RoboDK station: InvertedRobot.rdk

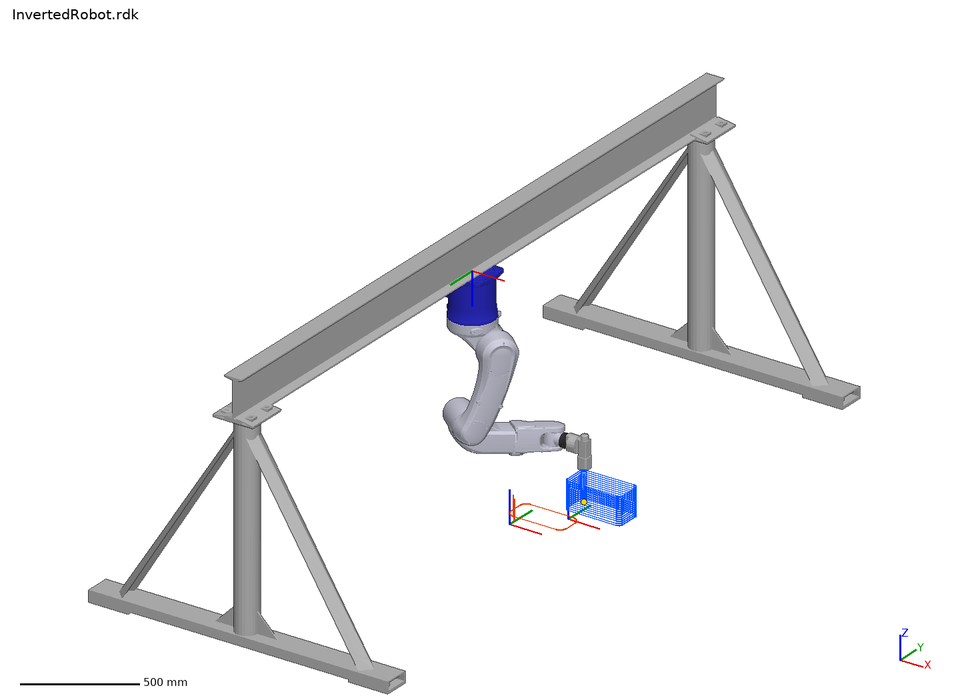
[picture v0: the station drawn from its stored meshes, robots at their saved joint values, targets as dots, program paths as lines]
Station InvertedRobot (saved by RoboDK 5.5.4). Poses are relative to the parent item; angles as X-Y-Z fixed-axis rotations.
Station parameters (name, value as stored): TAGS, ['Additive Manufacturing', 'Additive manufacturing']
  - frame Denso 1 at (0, -20, 974.25) mm, rotated rx -180 ry 0 rz 0 deg
    - robot Denso VS-6577G-B: 6 axes, payload 7 kg, reach 854 mm, repeatability 0.03 mm, weight 36 kg
        modified DH rows (alpha deg, a mm, theta deg, d mm): 0, 0, 0, 335; -90, 75, -90, 0; 0, 365, -90, 0; -90, 90, 0, 405; 90, 0, 0, 0; -90, 0, 0, 80
        joint limits [-170, -100, -119, -190, -120, -360] to [170, 135, 169, 190, 120, 360]; home [0, 0, 90, 0, 0, 0]; saved at [-52.91, -18.13, 101.16, 84.758, 53.229, -81.286]
      - tool nozzle, TCP at (110, 0, 80) mm, rotated rx 0 ry 90 rz 0 deg, size 158.8 x 76.2 x 114.9 mm, geometry from nozzle.STEP
  - frame Ref001 at (404.35, 97.88, -110) mm
    - object Part at (0, 0, 0) mm, size 120 x 120 x 160 mm, geometry from part.sld
  - machining project Print3D settings: C:/Users/silverBlacK/OneDrive - University of Idaho/Research/RoboticsResearch/WallSection.gcode | rotZ(0) | rotX(0)*rotY(0) | rotZ(0)
  - program Print3D1 (17608 instructions, listed below)
  - frame Ref002 at (374.35, -282.12, 10) mm
    - object Part at (0, 0, 0) mm, size 120 x 120 x 160 mm, geometry from part.sld
  - machining project Print3D settings: C:/Users/silverBlacK/OneDrive - University of Idaho/Research/RoboticsResearch/WallSections/12x12x0.875.gcode | rotZ(0) | rotX(0)*rotY(0) | rotz(0) | onStart | onPathStart | onApproach | onPoint | onRetract | onFinish | SetRPM(%1) | SetTool(%1) | Extruder(%1) | default | default | OutOnMov(%1) | OutOffMov(%1) | onPathFinish | M_RunCode(%1)
  - program Print3D (292 instructions, listed below)
  - Python program Extruder (listed below)
  - Python program SimulateFinalResult (listed below)
  - object GantryAssembly at (-570, -550, -380) mm, rotated rx 90 ry 0 rz 0 deg, size 1524 x 1270 x 3505.2 mm, geometry from GantryAssembly.STEP
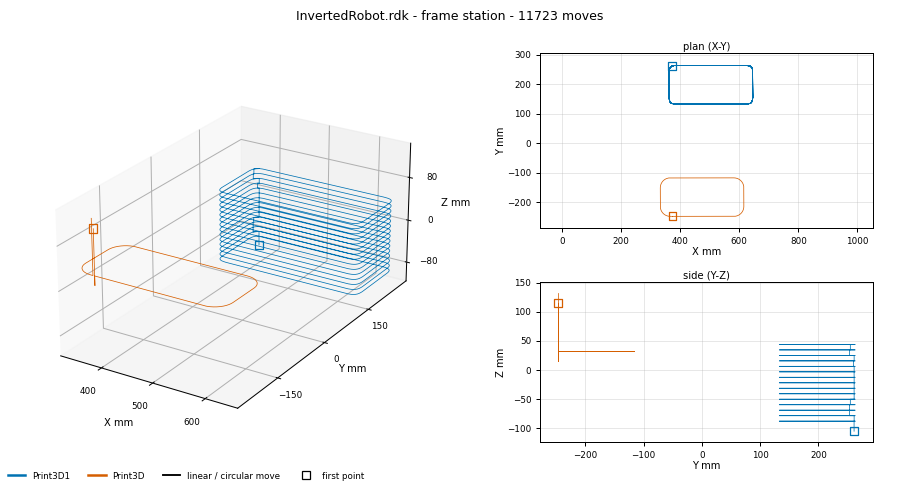
[picture p0: tool path of InvertedRobot.rdk in frame station, 11723 of 11723 moves have a stored position in this frame; points joined in program order, loops and branches not executed]

--- program Print3D1 (robot Denso VS-6577G-B) ---
  Smooth(1)
  Call M_RunCode(107)
  Call M_RunCode(104)
  Set speed (83.3 mm/s)
  Set speed (1000.0 mm/s)
  Set Ref.: Ref001
  Set Tool: nozzle
  Show nozzle
  MoveJ 1 to (-31.64, 163.21, 5) mm, rotated rx -180 ry 0 rz 180 deg; joints [-52.884, -5.749, 67.478, 70.281, 57.897, -56.003]
  MoveL 2 to (-31.64, 163.21, 5) mm, rotated rx -180 ry 0 rz 180 deg; joints [-52.884, -5.749, 67.478, 70.281, 57.897, -56.003]
  Call Extruder(-1)
  MoveL 3 to (-31.64, 163.21, 5) mm, rotated rx -180 ry 0 rz 180 deg; joints [-52.884, -5.749, 67.478, 70.281, 57.897, -56.003]
  Call M_RunCode(109)
  Call M_RunCode(82)
  Call Extruder(0.00000)
  Set speed (130.0 mm/s)
  MoveL 4 to (-31.64, 163.21, 22.23) mm, rotated rx 180 ry 0 rz -180 deg; joints [-52.884, -7.787, 72.321, 71.976, 56.989, -59.153]
  Call Extruder(-2.00000)
  Set speed (40.0 mm/s)
  MoveL 5 to (-31.64, 163.21, 22.23) mm, rotated rx 180 ry 0 rz -180 deg; joints [-52.884, -7.787, 72.321, 71.976, 56.989, -59.153]
  Call Extruder(0.00000)
  Set speed (130.0 mm/s)
  MoveL 6 to (-31.64, 163.21, 22.23) mm, rotated rx 180 ry 0 rz -180 deg; joints [-52.884, -7.787, 72.321, 71.976, 56.989, -59.153]
  Call Extruder(2.00000)
  Set speed (40.0 mm/s)
  MoveL 7 to (-31.64, 163.21, 22.23) mm, rotated rx 180 ry 0 rz -180 deg; joints [-52.884, -7.787, 72.321, 71.976, 56.989, -59.153]
  Set speed (30.0 mm/s)
  MoveL 8 to (-31.64, 163.21, 22.23) mm, rotated rx 180 ry 0 rz -180 deg; joints [-52.884, -7.787, 72.321, 71.976, 56.989, -59.153]
  Call Extruder(2.38024)
  MoveL 9 to (-31.93, 163.09, 22.22) mm, rotated rx 180 ry 0 rz 180 deg; joints [-52.91, -7.826, 72.354, 71.989, 57.013, -59.155]
  MoveL 10 to (-31.93, 163.09, 22.22) mm, rotated rx 180 ry 0 rz 180 deg; joints [-52.91, -7.826, 72.354, 71.989, 57.013, -59.155]
  Call Extruder(2.76227)
  MoveL 11 to (-32.22, 162.97, 22.22) mm, rotated rx 180 ry 0 rz -180 deg; joints [-52.936, -7.865, 72.387, 72.001, 57.037, -59.157]
  MoveL 12 to (-32.22, 162.97, 22.22) mm, rotated rx 180 ry 0 rz -180 deg; joints [-52.936, -7.865, 72.387, 72.001, 57.037, -59.157]
  Call Extruder(3.11872)
  MoveL 13 to (-32.49, 162.85, 22.22) mm, rotated rx -180 ry 0 rz 180 deg; joints [-52.96, -7.901, 72.418, 72.012, 57.06, -59.158]
  MoveL 14 to (-32.49, 162.85, 22.22) mm, rotated rx -180 ry 0 rz 180 deg; joints [-52.96, -7.901, 72.418, 72.012, 57.06, -59.158]
  Call Extruder(3.44932)
  MoveL 15 to (-32.74, 162.74, 22.22) mm, rotated rx 180 ry 0 rz 180 deg; joints [-52.982, -7.935, 72.446, 72.022, 57.08, -59.16]
  MoveL 16 to (-32.74, 162.74, 22.22) mm, rotated rx 180 ry 0 rz 180 deg; joints [-52.982, -7.935, 72.446, 72.022, 57.08, -59.16]
  Call Extruder(3.78134)
  MoveL 17 to (-32.99, 162.64, 22.22) mm, rotated rx -180 ry 0 rz 180 deg; joints [-53.004, -7.968, 72.475, 72.032, 57.1, -59.161]
  MoveL 18 to (-32.99, 162.64, 22.22) mm, rotated rx -180 ry 0 rz 180 deg; joints [-53.004, -7.968, 72.475, 72.032, 57.1, -59.161]
  Call Extruder(4.21321)
  MoveL 19 to (-33.29, 162.46, 22.22) mm, rotated rx -180 ry 0 rz 180 deg; joints [-53.026, -8.015, 72.514, 72.042, 57.122, -59.16]
  MoveL 20 to (-33.29, 162.46, 22.22) mm, rotated rx -180 ry 0 rz 180 deg; joints [-53.026, -8.015, 72.514, 72.042, 57.122, -59.16]
  Call Extruder(4.64692)
  MoveL 21 to (-33.6, 162.29, 22.22) mm, rotated rx 180 ry 0 rz 180 deg; joints [-53.049, -8.061, 72.553, 72.051, 57.143, -59.16]
  MoveL 22 to (-33.6, 162.29, 22.22) mm, rotated rx 180 ry 0 rz 180 deg; joints [-53.049, -8.061, 72.553, 72.051, 57.143, -59.16]
  Call Extruder(5.08247)
  MoveL 23 to (-33.9, 162.11, 22.23) mm, rotated rx 180 ry 0 rz 180 deg; joints [-53.071, -8.107, 72.591, 72.06, 57.165, -59.159]
  MoveL 24 to (-33.9, 162.11, 22.23) mm, rotated rx 180 ry 0 rz 180 deg; joints [-53.071, -8.107, 72.591, 72.06, 57.165, -59.159]
  Call Extruder(5.51986)
  MoveL 25 to (-34.21, 161.94, 22.22) mm, rotated rx 180 ry 0 rz 180 deg; joints [-53.094, -8.153, 72.63, 72.07, 57.186, -59.158]
  MoveL 26 to (-34.21, 161.94, 22.22) mm, rotated rx 180 ry 0 rz 180 deg; joints [-53.094, -8.153, 72.63, 72.07, 57.186, -59.158]
  Call Extruder(5.89660)
  MoveL 27 to (-34.45, 161.76, 22.22) mm, rotated rx 180 ry 0 rz 180 deg; joints [-53.109, -8.194, 72.665, 72.075, 57.201, -59.156]
  MoveL 28 to (-34.45, 161.76, 22.22) mm, rotated rx 180 ry 0 rz 180 deg; joints [-53.109, -8.194, 72.665, 72.075, 57.201, -59.156]
  Call Extruder(6.59657)
  MoveL 29 to (-34.9, 161.43, 22.23) mm, rotated rx 180 ry 0 rz 180 deg; joints [-53.135, -8.27, 72.728, 72.084, 57.228, -59.151]
  MoveL 30 to (-34.9, 161.43, 22.23) mm, rotated rx 180 ry 0 rz 180 deg; joints [-53.135, -8.27, 72.728, 72.084, 57.228, -59.151]
  Call Extruder(7.29934)
  MoveL 31 to (-35.35, 161.1, 22.22) mm, rotated rx 180 ry 0 rz 180 deg; joints [-53.163, -8.346, 72.792, 72.093, 57.255, -59.146]
  Call Extruder(9.03811)
  MoveL 32 to (-36.39, 160.19, 22.22) mm, rotated rx 180 ry 0 rz 180 deg; joints [-53.209, -8.538, 72.953, 72.102, 57.305, -59.126]
  Call Extruder(10.77694)
  MoveL 33 to (-37.3, 159.15, 22.22) mm, rotated rx 180 ry 0 rz 180 deg; joints [-53.227, -8.733, 73.115, 72.093, 57.33, -59.094]
  Call Extruder(11.12832)
  MoveL 34 to (-37.47, 158.93, 22.22) mm, rotated rx 180 ry 0 rz -180 deg; joints [-53.227, -8.773, 73.148, 72.088, 57.332, -59.087]
  MoveL 35 to (-37.47, 158.93, 22.22) mm, rotated rx 180 ry 0 rz -180 deg; joints [-53.227, -8.773, 73.148, 72.088, 57.332, -59.087]
  Call Extruder(11.82828)
  MoveL 36 to (-37.79, 158.48, 22.22) mm, rotated rx 180 ry 0 rz 180 deg; joints [-53.226, -8.852, 73.214, 72.079, 57.335, -59.071]
  MoveL 37 to (-37.79, 158.48, 22.22) mm, rotated rx 180 ry 0 rz 180 deg; joints [-53.226, -8.852, 73.214, 72.079, 57.335, -59.071]
  Call Extruder(12.52544)
  MoveL 38 to (-38.12, 158.03, 22.22) mm, rotated rx 180 ry 0 rz 180 deg; joints [-53.224, -8.931, 73.279, 72.07, 57.338, -59.055]
  MoveL 39 to (-38.12, 158.03, 22.22) mm, rotated rx 180 ry 0 rz 180 deg; joints [-53.224, -8.931, 73.279, 72.07, 57.338, -59.055]
  Call Extruder(12.77229)
  MoveL 40 to (-38.22, 157.85, 22.22) mm, rotated rx -180 ry 0 rz 180 deg; joints [-53.221, -8.959, 73.302, 72.065, 57.336, -59.048]
  MoveL 41 to (-38.22, 157.85, 22.22) mm, rotated rx -180 ry 0 rz 180 deg; joints [-53.221, -8.959, 73.302, 72.065, 57.336, -59.048]
  Call Extruder(13.20785)
  MoveL 42 to (-38.4, 157.55, 22.22) mm, rotated rx 180 ry 0 rz 180 deg; joints [-53.214, -9.008, 73.343, 72.055, 57.333, -59.036]
  MoveL 43 to (-38.4, 157.55, 22.22) mm, rotated rx 180 ry 0 rz 180 deg; joints [-53.214, -9.008, 73.343, 72.055, 57.333, -59.036]
  Call Extruder(13.64157)
  MoveL 44 to (-38.57, 157.25, 22.22) mm, rotated rx -180 ry 0 rz 180 deg; joints [-53.207, -9.057, 73.383, 72.046, 57.33, -59.024]
  MoveL 45 to (-38.57, 157.25, 22.22) mm, rotated rx -180 ry 0 rz 180 deg; joints [-53.207, -9.057, 73.383, 72.046, 57.33, -59.024]
  Call Extruder(14.07344)
  MoveL 46 to (-38.75, 156.94, 22.22) mm, rotated rx 180 ry 0 rz 180 deg; joints [-53.2, -9.106, 73.424, 72.036, 57.327, -59.012]
  MoveL 47 to (-38.75, 156.94, 22.22) mm, rotated rx 180 ry 0 rz 180 deg; joints [-53.2, -9.106, 73.424, 72.036, 57.327, -59.012]
  Call Extruder(14.45383)
  MoveL 48 to (-38.89, 156.67, 22.22) mm, rotated rx 180 ry 0 rz 180 deg; joints [-53.191, -9.15, 73.459, 72.026, 57.322, -59.001]
  MoveL 49 to (-38.89, 156.67, 22.22) mm, rotated rx 180 ry 0 rz 180 deg; joints [-53.191, -9.15, 73.459, 72.026, 57.322, -59.001]
  Call Extruder(14.78446)
  MoveL 50 to (-39, 156.42, 22.22) mm, rotated rx 180 ry 0 rz 180 deg; joints [-53.18, -9.187, 73.49, 72.016, 57.314, -58.99]
  MoveL 51 to (-39, 156.42, 22.22) mm, rotated rx 180 ry 0 rz 180 deg; joints [-53.18, -9.187, 73.49, 72.016, 57.314, -58.99]
  Call Extruder(15.11366)
  MoveL 52 to (-39.11, 156.17, 22.22) mm, rotated rx 180 ry 0 rz 180 deg; joints [-53.17, -9.224, 73.52, 72.005, 57.307, -58.979]
  MoveL 53 to (-39.11, 156.17, 22.22) mm, rotated rx 180 ry 0 rz 180 deg; joints [-53.17, -9.224, 73.52, 72.005, 57.307, -58.979]
  Call Extruder(15.49565)
  MoveL 54 to (-39.23, 155.88, 22.22) mm, rotated rx 180 ry 0 rz 180 deg; joints [-53.156, -9.267, 73.556, 71.992, 57.298, -58.965]
  MoveL 55 to (-39.23, 155.88, 22.22) mm, rotated rx 180 ry 0 rz 180 deg; joints [-53.156, -9.267, 73.556, 71.992, 57.298, -58.965]
  Call Extruder(15.87585)
  MoveL 56 to (-39.35, 155.58, 22.22) mm, rotated rx 180 ry 0 rz 180 deg; joints [-53.143, -9.31, 73.591, 71.98, 57.29, -58.952]
  MoveL 57 to (-39.35, 155.58, 22.22) mm, rotated rx 180 ry 0 rz 180 deg; joints [-53.143, -9.31, 73.591, 71.98, 57.29, -58.952]
  Call Extruder(16.18353)
  MoveL 58 to (-39.44, 155.34, 22.23) mm, rotated rx 180 ry 0 rz 180 deg; joints [-53.131, -9.345, 73.619, 71.968, 57.281, -58.941]
  MoveL 59 to (-39.44, 155.34, 22.23) mm, rotated rx 180 ry 0 rz 180 deg; joints [-53.131, -9.345, 73.619, 71.968, 57.281, -58.941]
  Call Extruder(16.41988)
  MoveL 60 to (-39.5, 155.15, 22.22) mm, rotated rx 180 ry 0 rz 180 deg; joints [-53.121, -9.371, 73.641, 71.959, 57.274, -58.932]
  MoveL 61 to (-39.5, 155.15, 22.22) mm, rotated rx 180 ry 0 rz 180 deg; joints [-53.121, -9.371, 73.641, 71.959, 57.274, -58.932]
  Call Extruder(16.65518)
  MoveL 62 to (-39.56, 154.97, 22.23) mm, rotated rx 180 ry 0 rz 180 deg; joints [-53.11, -9.398, 73.663, 71.949, 57.266, -58.923]
  MoveL 63 to (-39.56, 154.97, 22.23) mm, rotated rx 180 ry 0 rz 180 deg; joints [-53.11, -9.398, 73.663, 71.949, 57.266, -58.923]
  Call Extruder(16.88943)
  MoveL 64 to (-39.62, 154.78, 22.22) mm, rotated rx 180 ry 0 rz 180 deg; joints [-53.099, -9.424, 73.684, 71.94, 57.258, -58.914]
  MoveL 65 to (-39.62, 154.78, 22.22) mm, rotated rx 180 ry 0 rz 180 deg; joints [-53.099, -9.424, 73.684, 71.94, 57.258, -58.914]
  Call Extruder(17.12262)
  MoveL 66 to (-39.68, 154.59, 22.22) mm, rotated rx 180 ry 0 rz -180 deg; joints [-53.088, -9.45, 73.706, 71.93, 57.25, -58.905]
  MoveL 67 to (-39.68, 154.59, 22.22) mm, rotated rx 180 ry 0 rz -180 deg; joints [-53.088, -9.45, 73.706, 71.93, 57.25, -58.905]
  Call Extruder(17.37548)
  MoveL 68 to (-39.75, 154.38, 22.23) mm, rotated rx 180 ry 0 rz 180 deg; joints [-53.076, -9.479, 73.729, 71.919, 57.242, -58.895]
  MoveL 69 to (-39.75, 154.38, 22.23) mm, rotated rx 180 ry 0 rz 180 deg; joints [-53.076, -9.479, 73.729, 71.919, 57.242, -58.895]
  Call Extruder(17.64775)
  MoveL 70 to (-39.81, 154.16, 22.23) mm, rotated rx 180 ry 0 rz 180 deg; joints [-53.063, -9.51, 73.754, 71.908, 57.232, -58.884]
  MoveL 71 to (-39.81, 154.16, 22.23) mm, rotated rx 180 ry 0 rz 180 deg; joints [-53.063, -9.51, 73.754, 71.908, 57.232, -58.884]
  Call Extruder(17.91868)
  MoveL 72 to (-39.88, 153.94, 22.22) mm, rotated rx 180 ry 0 rz 180 deg; joints [-53.049, -9.541, 73.779, 71.896, 57.222, -58.873]
  MoveL 73 to (-39.88, 153.94, 22.22) mm, rotated rx 180 ry 0 rz 180 deg; joints [-53.049, -9.541, 73.779, 71.896, 57.222, -58.873]
  Call Extruder(18.18828)
  MoveL 74 to (-39.95, 153.71, 22.23) mm, rotated rx 180 ry 0 rz 180 deg; joints [-53.036, -9.572, 73.804, 71.884, 57.212, -58.862]
  MoveL 75 to (-39.95, 153.71, 22.23) mm, rotated rx 180 ry 0 rz 180 deg; joints [-53.036, -9.572, 73.804, 71.884, 57.212, -58.862]
  Call Extruder(18.45654)
  MoveL 76 to (-40.02, 153.49, 22.23) mm, rotated rx 180 ry 0 rz 180 deg; joints [-53.022, -9.602, 73.829, 71.872, 57.202, -58.851]
  MoveL 77 to (-40.02, 153.49, 22.23) mm, rotated rx 180 ry 0 rz 180 deg; joints [-53.022, -9.602, 73.829, 71.872, 57.202, -58.851]
  Call Extruder(18.69554)
  MoveL 78 to (-40.06, 153.28, 22.23) mm, rotated rx 180 ry 0 rz 180 deg; joints [-53.007, -9.629, 73.851, 71.86, 57.191, -58.841]
  MoveL 79 to (-40.06, 153.28, 22.23) mm, rotated rx 180 ry 0 rz 180 deg; joints [-53.007, -9.629, 73.851, 71.86, 57.191, -58.841]
  Call Extruder(18.93348)
  MoveL 80 to (-40.11, 153.08, 22.22) mm, rotated rx -180 ry 0 rz 180 deg; joints [-52.993, -9.656, 73.873, 71.848, 57.18, -58.83]
  MoveL 81 to (-40.11, 153.08, 22.22) mm, rotated rx -180 ry 0 rz 180 deg; joints [-52.993, -9.656, 73.873, 71.848, 57.18, -58.83]
  Call Extruder(19.17035)
  MoveL 82 to (-40.15, 152.88, 22.23) mm, rotated rx 180 ry 0 rz 180 deg; joints [-52.978, -9.682, 73.894, 71.836, 57.169, -58.819]
  MoveL 83 to (-40.15, 152.88, 22.23) mm, rotated rx 180 ry 0 rz 180 deg; joints [-52.978, -9.682, 73.894, 71.836, 57.169, -58.819]
  Call Extruder(19.40615)
  MoveL 84 to (-40.2, 152.67, 22.23) mm, rotated rx 180 ry 0 rz 180 deg; joints [-52.963, -9.709, 73.916, 71.824, 57.158, -58.809]
  MoveL 85 to (-40.2, 152.67, 22.23) mm, rotated rx 180 ry 0 rz 180 deg; joints [-52.963, -9.709, 73.916, 71.824, 57.158, -58.809]
  Call Extruder(19.66605)
  MoveL 86 to (-40.24, 152.45, 22.23) mm, rotated rx 180 ry 0 rz 180 deg; joints [-52.946, -9.738, 73.94, 71.81, 57.146, -58.797]
  MoveL 87 to (-40.24, 152.45, 22.23) mm, rotated rx 180 ry 0 rz 180 deg; joints [-52.946, -9.738, 73.94, 71.81, 57.146, -58.797]
  Call Extruder(19.94972)
  MoveL 88 to (-40.29, 152.2, 22.22) mm, rotated rx 180 ry 0 rz 180 deg; joints [-52.928, -9.77, 73.966, 71.795, 57.132, -58.784]
  MoveL 89 to (-40.29, 152.2, 22.22) mm, rotated rx 180 ry 0 rz 180 deg; joints [-52.928, -9.77, 73.966, 71.795, 57.132, -58.784]
  Call Extruder(20.23193)
  MoveL 90 to (-40.34, 151.95, 22.22) mm, rotated rx 180 ry 0 rz 180 deg; joints [-52.909, -9.803, 73.992, 71.779, 57.117, -58.77]
  MoveL 91 to (-40.34, 151.95, 22.22) mm, rotated rx 180 ry 0 rz 180 deg; joints [-52.909, -9.803, 73.992, 71.779, 57.117, -58.77]
  Call Extruder(20.51271)
  MoveL 92 to (-40.39, 151.7, 22.23) mm, rotated rx 180 ry 0 rz 180 deg; joints [-52.89, -9.835, 74.018, 71.764, 57.103, -58.757]
  MoveL 93 to (-40.39, 151.7, 22.23) mm, rotated rx 180 ry 0 rz 180 deg; joints [-52.89, -9.835, 74.018, 71.764, 57.103, -58.757]
  Call Extruder(20.79205)
  MoveL 94 to (-40.44, 151.45, 22.22) mm, rotated rx 180 ry 0 rz -180 deg; joints [-52.871, -9.867, 74.043, 71.748, 57.089, -58.744]
  MoveL 95 to (-40.44, 151.45, 22.22) mm, rotated rx 180 ry 0 rz -180 deg; joints [-52.871, -9.867, 74.043, 71.748, 57.089, -58.744]
  Call Extruder(21.06994)
  MoveL 96 to (-40.49, 151.2, 22.22) mm, rotated rx 180 ry 0 rz 180 deg; joints [-52.853, -9.899, 74.069, 71.733, 57.075, -58.731]
  MoveL 97 to (-40.49, 151.2, 22.22) mm, rotated rx 180 ry 0 rz 180 deg; joints [-52.853, -9.899, 74.069, 71.733, 57.075, -58.731]
  Call Extruder(21.34639)
  MoveL 98 to (-40.54, 150.95, 22.23) mm, rotated rx 180 ry 0 rz 180 deg; joints [-52.834, -9.93, 74.095, 71.718, 57.061, -58.717]
  MoveL 99 to (-40.54, 150.95, 22.23) mm, rotated rx 180 ry 0 rz 180 deg; joints [-52.834, -9.93, 74.095, 71.718, 57.061, -58.717]
  Call Extruder(21.65140)
  MoveL 100 to (-40.59, 150.67, 22.22) mm, rotated rx 180 ry 0 rz 180 deg; joints [-52.812, -9.966, 74.123, 71.7, 57.044, -58.702]
  MoveL 101 to (-40.59, 150.67, 22.22) mm, rotated rx 180 ry 0 rz 180 deg; joints [-52.812, -9.966, 74.123, 71.7, 57.044, -58.702]
  Call Extruder(21.98479)
  MoveL 102 to (-40.64, 150.37, 22.22) mm, rotated rx -180 ry 0 rz 180 deg; joints [-52.787, -10.004, 74.154, 71.68, 57.025, -58.686]
  MoveL 103 to (-40.64, 150.37, 22.22) mm, rotated rx -180 ry 0 rz 180 deg; joints [-52.787, -10.004, 74.154, 71.68, 57.025, -58.686]
  Call Extruder(22.31647)
  MoveL 104 to (-40.69, 150.06, 22.22) mm, rotated rx 180 ry 0 rz 180 deg; joints [-52.762, -10.042, 74.185, 71.66, 57.006, -58.669]
  MoveL 105 to (-40.69, 150.06, 22.22) mm, rotated rx 180 ry 0 rz 180 deg; joints [-52.762, -10.042, 74.185, 71.66, 57.006, -58.669]
  Call Extruder(22.64643)
  MoveL 106 to (-40.74, 149.76, 22.22) mm, rotated rx -180 ry 0 rz 180 deg; joints [-52.737, -10.08, 74.215, 71.64, 56.988, -58.652]
  MoveL 107 to (-40.74, 149.76, 22.22) mm, rotated rx -180 ry 0 rz 180 deg; joints [-52.737, -10.08, 74.215, 71.64, 56.988, -58.652]
  Call Extruder(22.97467)
  MoveL 108 to (-40.78, 149.45, 22.23) mm, rotated rx 180 ry 0 rz 180 deg; joints [-52.712, -10.118, 74.246, 71.62, 56.969, -58.635]
  MoveL 109 to (-40.78, 149.45, 22.23) mm, rotated rx 180 ry 0 rz 180 deg; joints [-52.712, -10.118, 74.246, 71.62, 56.969, -58.635]
  Call Extruder(23.30119)
  MoveL 110 to (-40.83, 149.14, 22.22) mm, rotated rx 180 ry 0 rz -180 deg; joints [-52.687, -10.156, 74.277, 71.6, 56.95, -58.618]
  MoveL 111 to (-40.83, 149.14, 22.22) mm, rotated rx 180 ry 0 rz -180 deg; joints [-52.687, -10.156, 74.277, 71.6, 56.95, -58.618]
  Call Extruder(23.66827)
  MoveL 112 to (-40.88, 148.8, 22.23) mm, rotated rx 180 ry 0 rz -180 deg; joints [-52.658, -10.199, 74.311, 71.576, 56.927, -58.598]
  MoveL 113 to (-40.88, 148.8, 22.23) mm, rotated rx 180 ry 0 rz -180 deg; joints [-52.658, -10.199, 74.311, 71.576, 56.927, -58.598]
  Call Extruder(24.07571)
  MoveL 114 to (-40.92, 148.41, 22.22) mm, rotated rx 180 ry 0 rz 180 deg; joints [-52.624, -10.246, 74.348, 71.549, 56.901, -58.576]
  MoveL 115 to (-40.92, 148.41, 22.22) mm, rotated rx 180 ry 0 rz 180 deg; joints [-52.624, -10.246, 74.348, 71.549, 56.901, -58.576]
  Call Extruder(24.48110)
  MoveL 116 to (-40.97, 148.02, 22.22) mm, rotated rx 180 ry 0 rz 180 deg; joints [-52.59, -10.292, 74.386, 71.522, 56.875, -58.554]
  MoveL 117 to (-40.97, 148.02, 22.22) mm, rotated rx 180 ry 0 rz 180 deg; joints [-52.59, -10.292, 74.386, 71.522, 56.875, -58.554]
  Call Extruder(24.88445)
  MoveL 118 to (-41.02, 147.63, 22.22) mm, rotated rx -180 ry 0 rz 180 deg; joints [-52.556, -10.339, 74.423, 71.495, 56.849, -58.532]
  MoveL 119 to (-41.02, 147.63, 22.22) mm, rotated rx -180 ry 0 rz 180 deg; joints [-52.556, -10.339, 74.423, 71.495, 56.849, -58.532]
  Call Extruder(25.28574)
  MoveL 120 to (-41.06, 147.25, 22.22) mm, rotated rx 180 ry 0 rz 180 deg; joints [-52.521, -10.386, 74.46, 71.468, 56.823, -58.51]
  MoveL 121 to (-41.06, 147.25, 22.22) mm, rotated rx 180 ry 0 rz 180 deg; joints [-52.521, -10.386, 74.46, 71.468, 56.823, -58.51]
  Call Extruder(25.89062)
  MoveL 122 to (-41.11, 146.66, 22.23) mm, rotated rx 180 ry 0 rz 180 deg; joints [-52.466, -10.455, 74.515, 71.425, 56.78, -58.475]
  MoveL 123 to (-41.11, 146.66, 22.23) mm, rotated rx 180 ry 0 rz 180 deg; joints [-52.466, -10.455, 74.515, 71.425, 56.78, -58.475]
  Call Extruder(26.49235)
  MoveL 124 to (-41.15, 146.07, 22.22) mm, rotated rx 180 ry 0 rz 180 deg; joints [-52.411, -10.524, 74.57, 71.381, 56.737, -58.44]
  MoveL 125 to (-41.15, 146.07, 22.22) mm, rotated rx 180 ry 0 rz 180 deg; joints [-52.411, -10.524, 74.57, 71.381, 56.737, -58.44]
  Call Extruder(27.09093)
  MoveL 126 to (-41.2, 145.48, 22.22) mm, rotated rx -180 ry 0 rz 180 deg; joints [-52.355, -10.593, 74.625, 71.338, 56.695, -58.404]
  MoveL 127 to (-41.2, 145.48, 22.22) mm, rotated rx -180 ry 0 rz 180 deg; joints [-52.355, -10.593, 74.625, 71.338, 56.695, -58.404]
  Call Extruder(28.26271)
  MoveL 128 to (-41.25, 144.32, 22.22) mm, rotated rx 180 ry 0 rz 180 deg; joints [-52.239, -10.724, 74.729, 71.247, 56.604, -58.333]
  MoveL 129 to (-41.25, 144.32, 22.22) mm, rotated rx 180 ry 0 rz 180 deg; joints [-52.239, -10.724, 74.729, 71.247, 56.604, -58.333]
  Call Extruder(29.72057)
  MoveL 130 to (-41.29, 142.86, 22.22) mm, rotated rx -180 ry 0 rz 180 deg; joints [-52.09, -10.887, 74.858, 71.132, 56.489, -58.243]
  Call Extruder(115.61408)
  MoveL 131 to (-41.29, 57.14, 22.22) mm, rotated rx 180 ry 0 rz 180 deg; joints [-40.759, -19.184, 80.692, 61.037, 48.262, -50.261]
  Call Extruder(116.48916)
  MoveL 132 to (-41.27, 56.26, 22.22) mm, rotated rx 180 ry 0 rz -180 deg; joints [-40.614, -19.255, 80.736, 60.892, 48.164, -50.147]
  MoveL 133 to (-41.27, 56.26, 22.22) mm, rotated rx 180 ry 0 rz -180 deg; joints [-40.614, -19.255, 80.736, 60.892, 48.164, -50.147]
  Call Extruder(117.66094)
  MoveL 134 to (-41.23, 55.1, 22.22) mm, rotated rx -180 ry 0 rz 180 deg; joints [-40.419, -19.347, 80.792, 60.696, 48.032, -49.993]
  MoveL 135 to (-41.23, 55.1, 22.22) mm, rotated rx -180 ry 0 rz 180 deg; joints [-40.419, -19.347, 80.792, 60.696, 48.032, -49.993]
  Call Extruder(118.54904)
  MoveL 136 to (-41.18, 54.23, 22.22) mm, rotated rx -180 ry 0 rz 180 deg; joints [-40.269, -19.414, 80.834, 60.545, 47.93, -49.875]
  MoveL 137 to (-41.18, 54.23, 22.22) mm, rotated rx -180 ry 0 rz 180 deg; joints [-40.269, -19.414, 80.834, 60.545, 47.93, -49.875]
  Call Extruder(119.15077)
  MoveL 138 to (-41.13, 53.64, 22.23) mm, rotated rx -180 ry 0 rz 180 deg; joints [-40.165, -19.458, 80.86, 60.442, 47.859, -49.794]
  MoveL 139 to (-41.13, 53.64, 22.23) mm, rotated rx -180 ry 0 rz 180 deg; joints [-40.165, -19.458, 80.86, 60.442, 47.859, -49.794]
  Call Extruder(119.75565)
  MoveL 140 to (-41.09, 53.05, 22.22) mm, rotated rx 180 ry 0 rz 180 deg; joints [-40.062, -19.502, 80.887, 60.338, 47.788, -49.714]
  MoveL 141 to (-41.09, 53.05, 22.22) mm, rotated rx 180 ry 0 rz 180 deg; joints [-40.062, -19.502, 80.887, 60.338, 47.788, -49.714]
  Call Extruder(120.26021)
  MoveL 142 to (-41.04, 52.56, 22.22) mm, rotated rx 180 ry 0 rz 180 deg; joints [-39.975, -19.538, 80.909, 60.251, 47.729, -49.646]
  MoveL 143 to (-41.04, 52.56, 22.22) mm, rotated rx 180 ry 0 rz 180 deg; joints [-39.975, -19.538, 80.909, 60.251, 47.729, -49.646]
  Call Extruder(120.66355)
  MoveL 144 to (-40.99, 52.17, 22.22) mm, rotated rx 180 ry 0 rz -180 deg; joints [-39.904, -19.565, 80.925, 60.181, 47.68, -49.592]
  MoveL 145 to (-40.99, 52.17, 22.22) mm, rotated rx 180 ry 0 rz -180 deg; joints [-39.904, -19.565, 80.925, 60.181, 47.68, -49.592]
  Call Extruder(121.06894)
  MoveL 146 to (-40.95, 51.78, 22.23) mm, rotated rx -180 ry 0 rz 180 deg; joints [-39.833, -19.592, 80.942, 60.111, 47.632, -49.538]
  MoveL 147 to (-40.95, 51.78, 22.23) mm, rotated rx -180 ry 0 rz 180 deg; joints [-39.833, -19.592, 80.942, 60.111, 47.632, -49.538]
  Call Extruder(121.47639)
  MoveL 148 to (-40.9, 51.4, 22.22) mm, rotated rx 180 ry 0 rz 180 deg; joints [-39.763, -19.619, 80.958, 60.04, 47.583, -49.484]
  MoveL 149 to (-40.9, 51.4, 22.22) mm, rotated rx 180 ry 0 rz 180 deg; joints [-39.763, -19.619, 80.958, 60.04, 47.583, -49.484]
  Call Extruder(121.88588)
  MoveL 150 to (-40.86, 51.01, 22.22) mm, rotated rx -180 ry 0 rz 180 deg; joints [-39.692, -19.646, 80.975, 59.969, 47.535, -49.429]
  MoveL 151 to (-40.86, 51.01, 22.22) mm, rotated rx -180 ry 0 rz 180 deg; joints [-39.692, -19.646, 80.975, 59.969, 47.535, -49.429]
  Call Extruder(122.21240)
  MoveL 152 to (-40.81, 50.7, 22.22) mm, rotated rx -180 ry 0 rz 180 deg; joints [-39.634, -19.666, 80.987, 59.912, 47.495, -49.386]
  MoveL 153 to (-40.81, 50.7, 22.22) mm, rotated rx -180 ry 0 rz 180 deg; joints [-39.634, -19.666, 80.987, 59.912, 47.495, -49.386]
  Call Extruder(122.54064)
  MoveL 154 to (-40.76, 50.4, 22.22) mm, rotated rx 180 ry 0 rz -180 deg; joints [-39.576, -19.686, 80.999, 59.854, 47.455, -49.342]
  MoveL 155 to (-40.76, 50.4, 22.22) mm, rotated rx 180 ry 0 rz -180 deg; joints [-39.576, -19.686, 80.999, 59.854, 47.455, -49.342]
  Call Extruder(122.87060)
  MoveL 156 to (-40.71, 50.09, 22.23) mm, rotated rx 180 ry 0 rz 180 deg; joints [-39.518, -19.706, 81.011, 59.797, 47.415, -49.298]
  MoveL 157 to (-40.71, 50.09, 22.23) mm, rotated rx 180 ry 0 rz 180 deg; joints [-39.518, -19.706, 81.011, 59.797, 47.415, -49.298]
  Call Extruder(123.20228)
  MoveL 158 to (-40.66, 49.79, 22.23) mm, rotated rx -180 ry 0 rz 180 deg; joints [-39.46, -19.726, 81.023, 59.74, 47.375, -49.254]
  MoveL 159 to (-40.66, 49.79, 22.23) mm, rotated rx -180 ry 0 rz 180 deg; joints [-39.46, -19.726, 81.023, 59.74, 47.375, -49.254]
  Call Extruder(123.53568)
  MoveL 160 to (-40.61, 49.48, 22.22) mm, rotated rx 180 ry 0 rz 180 deg; joints [-39.402, -19.746, 81.035, 59.682, 47.335, -49.21]
  MoveL 161 to (-40.61, 49.48, 22.22) mm, rotated rx 180 ry 0 rz 180 deg; joints [-39.402, -19.746, 81.035, 59.682, 47.335, -49.21]
  Call Extruder(123.87079)
  MoveL 162 to (-40.57, 49.17, 22.22) mm, rotated rx -180 ry 0 rz 180 deg; joints [-39.344, -19.765, 81.047, 59.624, 47.295, -49.166]
  MoveL 163 to (-40.57, 49.17, 22.22) mm, rotated rx -180 ry 0 rz 180 deg; joints [-39.344, -19.765, 81.047, 59.624, 47.295, -49.166]
  Call Extruder(124.14680)
  MoveL 164 to (-40.52, 48.93, 22.23) mm, rotated rx 180 ry 0 rz 180 deg; joints [-39.296, -19.781, 81.056, 59.576, 47.262, -49.129]
  MoveL 165 to (-40.52, 48.93, 22.23) mm, rotated rx 180 ry 0 rz 180 deg; joints [-39.296, -19.781, 81.056, 59.576, 47.262, -49.129]
  Call Extruder(124.42424)
  MoveL 166 to (-40.47, 48.68, 22.22) mm, rotated rx 180 ry 0 rz 180 deg; joints [-39.247, -19.796, 81.065, 59.528, 47.228, -49.093]
  MoveL 167 to (-40.47, 48.68, 22.22) mm, rotated rx 180 ry 0 rz 180 deg; joints [-39.247, -19.796, 81.065, 59.528, 47.228, -49.093]
  Call Extruder(124.70312)
  MoveL 168 to (-40.42, 48.43, 22.23) mm, rotated rx 180 ry 0 rz 180 deg; joints [-39.198, -19.811, 81.074, 59.479, 47.194, -49.056]
  MoveL 169 to (-40.42, 48.43, 22.23) mm, rotated rx 180 ry 0 rz 180 deg; joints [-39.198, -19.811, 81.074, 59.479, 47.194, -49.056]
  Call Extruder(124.98344)
  MoveL 170 to (-40.37, 48.18, 22.23) mm, rotated rx -180 ry 0 rz 180 deg; joints [-39.149, -19.826, 81.083, 59.431, 47.16, -49.019]
  MoveL 171 to (-40.37, 48.18, 22.23) mm, rotated rx -180 ry 0 rz 180 deg; joints [-39.149, -19.826, 81.083, 59.431, 47.16, -49.019]
  Call Extruder(125.26519)
  MoveL 172 to (-40.32, 47.93, 22.22) mm, rotated rx -180 ry 0 rz -180 deg; joints [-39.101, -19.841, 81.093, 59.382, 47.126, -48.983]
  MoveL 173 to (-40.32, 47.93, 22.22) mm, rotated rx -180 ry 0 rz -180 deg; joints [-39.101, -19.841, 81.093, 59.382, 47.126, -48.983]
  Call Extruder(125.54838)
  MoveL 174 to (-40.27, 47.68, 22.22) mm, rotated rx 180 ry 0 rz 180 deg; joints [-39.052, -19.856, 81.102, 59.334, 47.092, -48.946]
  MoveL 175 to (-40.27, 47.68, 22.22) mm, rotated rx 180 ry 0 rz 180 deg; joints [-39.052, -19.856, 81.102, 59.334, 47.092, -48.946]
  Call Extruder(125.76334)
  MoveL 176 to (-40.23, 47.49, 22.22) mm, rotated rx 180 ry 0 rz 180 deg; joints [-39.015, -19.867, 81.108, 59.297, 47.067, -48.918]
  MoveL 177 to (-40.23, 47.49, 22.22) mm, rotated rx 180 ry 0 rz 180 deg; joints [-39.015, -19.867, 81.108, 59.297, 47.067, -48.918]
  Call Extruder(125.95387)
  MoveL 178 to (-40.2, 47.33, 22.22) mm, rotated rx -180 ry 0 rz 180 deg; joints [-38.982, -19.877, 81.114, 59.265, 47.044, -48.893]
  MoveL 179 to (-40.2, 47.33, 22.22) mm, rotated rx -180 ry 0 rz 180 deg; joints [-38.982, -19.877, 81.114, 59.265, 47.044, -48.893]
  Call Extruder(126.19017)
  MoveL 180 to (-40.15, 47.12, 22.22) mm, rotated rx 180 ry 0 rz 180 deg; joints [-38.941, -19.889, 81.121, 59.224, 47.016, -48.863]
  MoveL 181 to (-40.15, 47.12, 22.22) mm, rotated rx 180 ry 0 rz 180 deg; joints [-38.941, -19.889, 81.121, 59.224, 47.016, -48.863]
  Call Extruder(126.42754)
  MoveL 182 to (-40.11, 46.92, 22.22) mm, rotated rx -180 ry 0 rz 180 deg; joints [-38.9, -19.901, 81.129, 59.184, 46.987, -48.832]
  MoveL 183 to (-40.11, 46.92, 22.22) mm, rotated rx -180 ry 0 rz 180 deg; joints [-38.9, -19.901, 81.129, 59.184, 46.987, -48.832]
  Call Extruder(126.66598)
  MoveL 184 to (-40.06, 46.72, 22.23) mm, rotated rx 180 ry 0 rz 180 deg; joints [-38.859, -19.912, 81.136, 59.143, 46.959, -48.802]
  MoveL 185 to (-40.06, 46.72, 22.23) mm, rotated rx 180 ry 0 rz 180 deg; joints [-38.859, -19.912, 81.136, 59.143, 46.959, -48.802]
  Call Extruder(126.90549)
  MoveL 186 to (-40.02, 46.51, 22.22) mm, rotated rx 180 ry 0 rz -180 deg; joints [-38.819, -19.924, 81.143, 59.102, 46.931, -48.771]
  MoveL 187 to (-40.02, 46.51, 22.22) mm, rotated rx 180 ry 0 rz -180 deg; joints [-38.819, -19.924, 81.143, 59.102, 46.931, -48.771]
  Call Extruder(127.17442)
  MoveL 188 to (-39.95, 46.29, 22.22) mm, rotated rx -180 ry 0 rz 180 deg; joints [-38.771, -19.935, 81.149, 59.056, 46.897, -48.736]
  MoveL 189 to (-39.95, 46.29, 22.22) mm, rotated rx -180 ry 0 rz 180 deg; joints [-38.771, -19.935, 81.149, 59.056, 46.897, -48.736]
  Call Extruder(127.44468)
  MoveL 190 to (-39.88, 46.06, 22.22) mm, rotated rx 180 ry 0 rz 180 deg; joints [-38.724, -19.946, 81.156, 59.01, 46.864, -48.702]
  MoveL 191 to (-39.88, 46.06, 22.22) mm, rotated rx 180 ry 0 rz 180 deg; joints [-38.724, -19.946, 81.156, 59.01, 46.864, -48.702]
  Call Extruder(127.71628)
  MoveL 192 to (-39.82, 45.84, 22.22) mm, rotated rx -180 ry 0 rz 180 deg; joints [-38.677, -19.957, 81.163, 58.963, 46.831, -48.668]
  MoveL 193 to (-39.82, 45.84, 22.22) mm, rotated rx -180 ry 0 rz 180 deg; joints [-38.677, -19.957, 81.163, 58.963, 46.831, -48.668]
  Call Extruder(127.98921)
  MoveL 194 to (-39.75, 45.62, 22.22) mm, rotated rx 180 ry 0 rz 180 deg; joints [-38.629, -19.968, 81.169, 58.917, 46.797, -48.633]
  MoveL 195 to (-39.75, 45.62, 22.22) mm, rotated rx 180 ry 0 rz 180 deg; joints [-38.629, -19.968, 81.169, 58.917, 46.797, -48.633]
  Call Extruder(128.24265)
  MoveL 196 to (-39.68, 45.41, 22.23) mm, rotated rx -180 ry 0 rz 180 deg; joints [-38.585, -19.978, 81.175, 58.874, 46.766, -48.601]
  MoveL 197 to (-39.68, 45.41, 22.23) mm, rotated rx -180 ry 0 rz 180 deg; joints [-38.585, -19.978, 81.175, 58.874, 46.766, -48.601]
  Call Extruder(128.47637)
  MoveL 198 to (-39.62, 45.22, 22.22) mm, rotated rx 180 ry 0 rz 180 deg; joints [-38.544, -19.987, 81.18, 58.834, 46.738, -48.572]
  MoveL 199 to (-39.62, 45.22, 22.22) mm, rotated rx 180 ry 0 rz 180 deg; joints [-38.544, -19.987, 81.18, 58.834, 46.738, -48.572]
  Call Extruder(128.71114)
  MoveL 200 to (-39.56, 45.03, 22.23) mm, rotated rx 180 ry 0 rz 180 deg; joints [-38.504, -19.996, 81.186, 58.794, 46.709, -48.542]
  MoveL 201 to (-39.56, 45.03, 22.23) mm, rotated rx 180 ry 0 rz 180 deg; joints [-38.504, -19.996, 81.186, 58.794, 46.709, -48.542]
  Call Extruder(128.94697)
  MoveL 202 to (-39.5, 44.85, 22.22) mm, rotated rx 180 ry 0 rz -180 deg; joints [-38.463, -20.005, 81.191, 58.754, 46.681, -48.513]
  MoveL 203 to (-39.5, 44.85, 22.22) mm, rotated rx 180 ry 0 rz -180 deg; joints [-38.463, -20.005, 81.191, 58.754, 46.681, -48.513]
  Call Extruder(129.18384)
  MoveL 204 to (-39.44, 44.66, 22.22) mm, rotated rx 180 ry 0 rz 180 deg; joints [-38.422, -20.013, 81.196, 58.714, 46.652, -48.483]
  MoveL 205 to (-39.44, 44.66, 22.22) mm, rotated rx 180 ry 0 rz 180 deg; joints [-38.422, -20.013, 81.196, 58.714, 46.652, -48.483]
  Call Extruder(129.49225)
  MoveL 206 to (-39.35, 44.42, 22.22) mm, rotated rx 180 ry 0 rz 180 deg; joints [-38.369, -20.023, 81.202, 58.662, 46.614, -48.445]
  MoveL 207 to (-39.35, 44.42, 22.22) mm, rotated rx 180 ry 0 rz 180 deg; joints [-38.369, -20.023, 81.202, 58.662, 46.614, -48.445]
  Call Extruder(129.87335)
  MoveL 208 to (-39.22, 44.12, 22.22) mm, rotated rx -180 ry 0 rz 180 deg; joints [-38.302, -20.034, 81.209, 58.598, 46.566, -48.398]
  MoveL 209 to (-39.22, 44.12, 22.22) mm, rotated rx -180 ry 0 rz 180 deg; joints [-38.302, -20.034, 81.209, 58.598, 46.566, -48.398]
  Call Extruder(130.25623)
  MoveL 210 to (-39.11, 43.83, 22.22) mm, rotated rx 180 ry 0 rz 180 deg; joints [-38.236, -20.045, 81.215, 58.533, 46.519, -48.351]
  MoveL 211 to (-39.11, 43.83, 22.22) mm, rotated rx 180 ry 0 rz 180 deg; joints [-38.236, -20.045, 81.215, 58.533, 46.519, -48.351]
  Call Extruder(130.58614)
  MoveL 212 to (-39, 43.58, 22.22) mm, rotated rx 180 ry 0 rz -180 deg; joints [-38.178, -20.054, 81.22, 58.478, 46.478, -48.31]
  MoveL 213 to (-39, 43.58, 22.22) mm, rotated rx 180 ry 0 rz -180 deg; joints [-38.178, -20.054, 81.22, 58.478, 46.478, -48.31]
  Call Extruder(130.91747)
  MoveL 214 to (-38.89, 43.33, 22.22) mm, rotated rx -180 ry 0 rz 180 deg; joints [-38.121, -20.063, 81.226, 58.422, 46.437, -48.27]
  MoveL 215 to (-38.89, 43.33, 22.22) mm, rotated rx -180 ry 0 rz 180 deg; joints [-38.121, -20.063, 81.226, 58.422, 46.437, -48.27]
  Call Extruder(131.29867)
  MoveL 216 to (-38.75, 43.06, 22.22) mm, rotated rx -180 ry 0 rz 180 deg; joints [-38.054, -20.07, 81.23, 58.358, 46.388, -48.224]
  MoveL 217 to (-38.75, 43.06, 22.22) mm, rotated rx -180 ry 0 rz 180 deg; joints [-38.054, -20.07, 81.23, 58.358, 46.388, -48.224]
  Call Extruder(131.73146)
  MoveL 218 to (-38.57, 42.75, 22.22) mm, rotated rx 180 ry 0 rz 180 deg; joints [-37.977, -20.076, 81.234, 58.286, 46.333, -48.172]
  MoveL 219 to (-38.57, 42.75, 22.22) mm, rotated rx 180 ry 0 rz 180 deg; joints [-37.977, -20.076, 81.234, 58.286, 46.333, -48.172]
  Call Extruder(132.16610)
  MoveL 220 to (-38.4, 42.45, 22.22) mm, rotated rx 180 ry 0 rz 180 deg; joints [-37.901, -20.083, 81.238, 58.214, 46.277, -48.121]
  MoveL 221 to (-38.4, 42.45, 22.22) mm, rotated rx 180 ry 0 rz 180 deg; joints [-37.901, -20.083, 81.238, 58.214, 46.277, -48.121]
  Call Extruder(132.60257)
  MoveL 222 to (-38.22, 42.15, 22.22) mm, rotated rx 180 ry 0 rz 180 deg; joints [-37.825, -20.089, 81.241, 58.141, 46.222, -48.069]
  MoveL 223 to (-38.22, 42.15, 22.22) mm, rotated rx 180 ry 0 rz 180 deg; joints [-37.825, -20.089, 81.241, 58.141, 46.222, -48.069]
  Call Extruder(132.84952)
  MoveL 224 to (-38.12, 41.98, 22.22) mm, rotated rx 180 ry 0 rz 180 deg; joints [-37.782, -20.092, 81.243, 58.1, 46.19, -48.04]
  MoveL 225 to (-38.12, 41.98, 22.22) mm, rotated rx 180 ry 0 rz 180 deg; joints [-37.782, -20.092, 81.243, 58.1, 46.19, -48.04]
  Call Extruder(133.54809)
  MoveL 226 to (-37.8, 41.52, 22.22) mm, rotated rx 180 ry 0 rz 180 deg; joints [-37.659, -20.094, 81.244, 57.985, 46.1, -47.96]
  MoveL 227 to (-37.8, 41.52, 22.22) mm, rotated rx 180 ry 0 rz 180 deg; joints [-37.659, -20.094, 81.244, 57.985, 46.1, -47.96]
  Call Extruder(134.24946)
  MoveL 228 to (-37.47, 41.07, 22.23) mm, rotated rx -180 ry 0 rz 180 deg; joints [-37.537, -20.096, 81.246, 57.871, 46.009, -47.88]
  MoveL 229 to (-37.47, 41.07, 22.23) mm, rotated rx -180 ry 0 rz 180 deg; joints [-37.537, -20.096, 81.246, 57.871, 46.009, -47.88]
  Call Extruder(134.60151)
  MoveL 230 to (-37.3, 40.85, 22.22) mm, rotated rx -180 ry 0 rz -180 deg; joints [-37.475, -20.097, 81.246, 57.813, 45.964, -47.84]
  Call Extruder(136.34360)
  MoveL 231 to (-36.39, 39.81, 22.22) mm, rotated rx 180 ry 0 rz 180 deg; joints [-37.173, -20.085, 81.239, 57.534, 45.737, -47.648]
  Call Extruder(137.66925)
  MoveL 232 to (-35.61, 39.11, 22.22) mm, rotated rx -180 ry 0 rz 180 deg; joints [-36.947, -20.059, 81.223, 57.329, 45.565, -47.511]
  MoveL 233 to (-35.61, 39.11, 22.22) mm, rotated rx -180 ry 0 rz 180 deg; joints [-36.947, -20.059, 81.223, 57.329, 45.565, -47.511]
  Call Extruder(138.08410)
  MoveL 234 to (-35.35, 38.9, 22.22) mm, rotated rx 180 ry 0 rz 180 deg; joints [-36.876, -20.05, 81.218, 57.265, 45.511, -47.469]
  Call Extruder(138.78545)
  MoveL 235 to (-34.9, 38.57, 22.22) mm, rotated rx 180 ry 0 rz -180 deg; joints [-36.759, -20.029, 81.205, 57.161, 45.42, -47.401]
  MoveL 236 to (-34.9, 38.57, 22.22) mm, rotated rx 180 ry 0 rz -180 deg; joints [-36.759, -20.029, 81.205, 57.161, 45.42, -47.401]
  Call Extruder(139.48400)
  MoveL 237 to (-34.45, 38.24, 22.22) mm, rotated rx -180 ry 0 rz -180 deg; joints [-36.642, -20.008, 81.193, 57.057, 45.33, -47.333]
  MoveL 238 to (-34.45, 38.24, 22.22) mm, rotated rx -180 ry 0 rz -180 deg; joints [-36.642, -20.008, 81.193, 57.057, 45.33, -47.333]
  Call Extruder(139.86003)
  MoveL 239 to (-34.21, 38.07, 22.22) mm, rotated rx 180 ry 0 rz 180 deg; joints [-36.579, -19.996, 81.186, 57.001, 45.281, -47.296]
  MoveL 240 to (-34.21, 38.07, 22.22) mm, rotated rx 180 ry 0 rz 180 deg; joints [-36.579, -19.996, 81.186, 57.001, 45.281, -47.296]
  Call Extruder(140.29650)
  MoveL 241 to (-33.9, 37.89, 22.23) mm, rotated rx 180 ry 0 rz 180 deg; joints [-36.509, -19.978, 81.175, 56.94, 45.225, -47.257]
  MoveL 242 to (-33.9, 37.89, 22.23) mm, rotated rx 180 ry 0 rz 180 deg; joints [-36.509, -19.978, 81.175, 56.94, 45.225, -47.257]
  Call Extruder(140.73113)
  MoveL 243 to (-33.6, 37.71, 22.23) mm, rotated rx 180 ry 0 rz 180 deg; joints [-36.439, -19.961, 81.165, 56.878, 45.17, -47.218]
  MoveL 244 to (-33.6, 37.71, 22.23) mm, rotated rx 180 ry 0 rz 180 deg; joints [-36.439, -19.961, 81.165, 56.878, 45.17, -47.218]
  Call Extruder(141.16391)
  MoveL 245 to (-33.29, 37.54, 22.23) mm, rotated rx 180 ry 0 rz 180 deg; joints [-36.368, -19.943, 81.154, 56.817, 45.114, -47.179]
  MoveL 246 to (-33.29, 37.54, 22.23) mm, rotated rx 180 ry 0 rz 180 deg; joints [-36.368, -19.943, 81.154, 56.817, 45.114, -47.179]
  Call Extruder(141.59485)
  MoveL 247 to (-32.99, 37.36, 22.22) mm, rotated rx -180 ry 0 rz 180 deg; joints [-36.298, -19.925, 81.143, 56.755, 45.059, -47.14]
  MoveL 248 to (-32.99, 37.36, 22.22) mm, rotated rx -180 ry 0 rz 180 deg; joints [-36.298, -19.925, 81.143, 56.755, 45.059, -47.14]
  Call Extruder(141.92621)
  MoveL 249 to (-32.74, 37.26, 22.22) mm, rotated rx 180 ry 0 rz 180 deg; joints [-36.247, -19.907, 81.133, 56.712, 45.017, -47.113]
  MoveL 250 to (-32.74, 37.26, 22.22) mm, rotated rx 180 ry 0 rz 180 deg; joints [-36.247, -19.907, 81.133, 56.712, 45.017, -47.113]
  Call Extruder(142.25615)
  MoveL 251 to (-32.49, 37.15, 22.22) mm, rotated rx -180 ry 0 rz 180 deg; joints [-36.196, -19.89, 81.122, 56.669, 44.976, -47.087]
  MoveL 252 to (-32.49, 37.15, 22.22) mm, rotated rx -180 ry 0 rz 180 deg; joints [-36.196, -19.89, 81.122, 56.669, 44.976, -47.087]
  Call Extruder(142.61184)
  MoveL 253 to (-32.22, 37.04, 22.23) mm, rotated rx 180 ry 0 rz 180 deg; joints [-36.141, -19.871, 81.111, 56.622, 44.932, -47.058]
  MoveL 254 to (-32.22, 37.04, 22.23) mm, rotated rx 180 ry 0 rz 180 deg; joints [-36.141, -19.871, 81.111, 56.622, 44.932, -47.058]
  Call Extruder(142.99292)
  MoveL 255 to (-31.93, 36.91, 22.22) mm, rotated rx -180 ry 0 rz 180 deg; joints [-36.082, -19.85, 81.098, 56.572, 44.884, -47.028]
  MoveL 256 to (-31.93, 36.91, 22.22) mm, rotated rx -180 ry 0 rz 180 deg; joints [-36.082, -19.85, 81.098, 56.572, 44.884, -47.028]
  Call Extruder(143.37221)
  MoveL 257 to (-31.64, 36.79, 22.22) mm, rotated rx 180 ry 0 rz 180 deg; joints [-36.023, -19.829, 81.086, 56.522, 44.837, -46.997]
  MoveL 258 to (-31.64, 36.79, 22.22) mm, rotated rx 180 ry 0 rz 180 deg; joints [-36.023, -19.829, 81.086, 56.522, 44.837, -46.997]
  Call Extruder(143.60909)
  MoveL 259 to (-31.45, 36.73, 22.22) mm, rotated rx 180 ry 0 rz 180 deg; joints [-35.989, -19.814, 81.077, 56.494, 44.808, -46.98]
  MoveL 260 to (-31.45, 36.73, 22.22) mm, rotated rx 180 ry 0 rz 180 deg; joints [-35.989, -19.814, 81.077, 56.494, 44.808, -46.98]
  Call Extruder(143.84491)
  MoveL 261 to (-31.26, 36.67, 22.23) mm, rotated rx -180 ry 0 rz -180 deg; joints [-35.954, -19.8, 81.068, 56.465, 44.779, -46.963]
  MoveL 262 to (-31.26, 36.67, 22.23) mm, rotated rx -180 ry 0 rz -180 deg; joints [-35.954, -19.8, 81.068, 56.465, 44.779, -46.963]
  Call Extruder(144.07969)
  MoveL 263 to (-31.07, 36.61, 22.22) mm, rotated rx 180 ry 0 rz 180 deg; joints [-35.919, -19.785, 81.059, 56.436, 44.751, -46.946]
  MoveL 264 to (-31.07, 36.61, 22.22) mm, rotated rx 180 ry 0 rz 180 deg; joints [-35.919, -19.785, 81.059, 56.436, 44.751, -46.946]
  Call Extruder(144.31341)
  MoveL 265 to (-30.88, 36.55, 22.22) mm, rotated rx -180 ry 0 rz 180 deg; joints [-35.884, -19.77, 81.05, 56.407, 44.722, -46.929]
  MoveL 266 to (-30.88, 36.55, 22.22) mm, rotated rx -180 ry 0 rz 180 deg; joints [-35.884, -19.77, 81.05, 56.407, 44.722, -46.929]
  Call Extruder(144.54609)
  MoveL 267 to (-30.69, 36.49, 22.22) mm, rotated rx 180 ry 0 rz 180 deg; joints [-35.849, -19.755, 81.041, 56.378, 44.693, -46.912]
  MoveL 268 to (-30.69, 36.49, 22.22) mm, rotated rx 180 ry 0 rz 180 deg; joints [-35.849, -19.755, 81.041, 56.378, 44.693, -46.912]
  Call Extruder(144.81901)
  MoveL 269 to (-30.47, 36.42, 22.22) mm, rotated rx -180 ry 0 rz 180 deg; joints [-35.809, -19.737, 81.03, 56.345, 44.66, -46.893]
  MoveL 270 to (-30.47, 36.42, 22.22) mm, rotated rx -180 ry 0 rz 180 deg; joints [-35.809, -19.737, 81.03, 56.345, 44.66, -46.893]
  Call Extruder(145.09061)
  MoveL 271 to (-30.25, 36.35, 22.22) mm, rotated rx 180 ry 0 rz 180 deg; joints [-35.768, -19.719, 81.019, 56.312, 44.626, -46.873]
  MoveL 272 to (-30.25, 36.35, 22.22) mm, rotated rx 180 ry 0 rz 180 deg; joints [-35.768, -19.719, 81.019, 56.312, 44.626, -46.873]
  Call Extruder(145.36086)
  MoveL 273 to (-30.02, 36.28, 22.22) mm, rotated rx -180 ry 0 rz 180 deg; joints [-35.728, -19.701, 81.008, 56.278, 44.593, -46.854]
  MoveL 274 to (-30.02, 36.28, 22.22) mm, rotated rx -180 ry 0 rz 180 deg; joints [-35.728, -19.701, 81.008, 56.278, 44.593, -46.854]
  Call Extruder(145.62979)
  MoveL 275 to (-29.8, 36.22, 22.22) mm, rotated rx 180 ry 0 rz -180 deg; joints [-35.688, -19.683, 80.997, 56.245, 44.56, -46.834]
  MoveL 276 to (-29.8, 36.22, 22.22) mm, rotated rx 180 ry 0 rz -180 deg; joints [-35.688, -19.683, 80.997, 56.245, 44.56, -46.834]
  Call Extruder(145.88314)
  MoveL 277 to (-29.59, 36.16, 22.22) mm, rotated rx -180 ry 0 rz 180 deg; joints [-35.651, -19.665, 80.986, 56.215, 44.529, -46.817]
  MoveL 278 to (-29.59, 36.16, 22.22) mm, rotated rx -180 ry 0 rz 180 deg; joints [-35.651, -19.665, 80.986, 56.215, 44.529, -46.817]
  Call Extruder(146.12159)
  MoveL 279 to (-29.38, 36.12, 22.23) mm, rotated rx 180 ry 0 rz 180 deg; joints [-35.617, -19.648, 80.976, 56.188, 44.501, -46.802]
  MoveL 280 to (-29.38, 36.12, 22.23) mm, rotated rx 180 ry 0 rz 180 deg; joints [-35.617, -19.648, 80.976, 56.188, 44.501, -46.802]
  Call Extruder(146.35896)
  MoveL 281 to (-29.18, 36.07, 22.22) mm, rotated rx -180 ry 0 rz 180 deg; joints [-35.584, -19.63, 80.965, 56.161, 44.472, -46.787]
  MoveL 282 to (-29.18, 36.07, 22.22) mm, rotated rx -180 ry 0 rz 180 deg; joints [-35.584, -19.63, 80.965, 56.161, 44.472, -46.787]
  Call Extruder(146.59526)
  MoveL 283 to (-28.97, 36.03, 22.22) mm, rotated rx -180 ry 0 rz 180 deg; joints [-35.55, -19.612, 80.954, 56.134, 44.444, -46.771]
  MoveL 284 to (-28.97, 36.03, 22.22) mm, rotated rx -180 ry 0 rz 180 deg; joints [-35.55, -19.612, 80.954, 56.134, 44.444, -46.771]
  Call Extruder(146.83050)
  MoveL 285 to (-28.77, 35.98, 22.22) mm, rotated rx 180 ry 0 rz -180 deg; joints [-35.517, -19.594, 80.943, 56.107, 44.415, -46.756]
  MoveL 286 to (-28.77, 35.98, 22.22) mm, rotated rx 180 ry 0 rz -180 deg; joints [-35.517, -19.594, 80.943, 56.107, 44.415, -46.756]
  Call Extruder(147.11443)
  MoveL 287 to (-28.52, 35.93, 22.22) mm, rotated rx 180 ry 0 rz 180 deg; joints [-35.477, -19.572, 80.93, 56.076, 44.381, -46.739]
  MoveL 288 to (-28.52, 35.93, 22.22) mm, rotated rx 180 ry 0 rz 180 deg; joints [-35.477, -19.572, 80.93, 56.076, 44.381, -46.739]
  Call Extruder(147.39692)
  MoveL 289 to (-28.27, 35.88, 22.22) mm, rotated rx 180 ry 0 rz 180 deg; joints [-35.437, -19.55, 80.916, 56.044, 44.348, -46.721]
  MoveL 290 to (-28.27, 35.88, 22.22) mm, rotated rx 180 ry 0 rz 180 deg; joints [-35.437, -19.55, 80.916, 56.044, 44.348, -46.721]
  Call Extruder(147.67798)
  MoveL 291 to (-28.02, 35.83, 22.22) mm, rotated rx 180 ry 0 rz 180 deg; joints [-35.397, -19.528, 80.903, 56.012, 44.314, -46.703]
  MoveL 292 to (-28.02, 35.83, 22.22) mm, rotated rx 180 ry 0 rz 180 deg; joints [-35.397, -19.528, 80.903, 56.012, 44.314, -46.703]
  Call Extruder(147.95760)
  MoveL 293 to (-27.77, 35.78, 22.22) mm, rotated rx -180 ry 0 rz -180 deg; joints [-35.357, -19.506, 80.889, 55.98, 44.28, -46.686]
  MoveL 294 to (-27.77, 35.78, 22.22) mm, rotated rx -180 ry 0 rz -180 deg; joints [-35.357, -19.506, 80.889, 55.98, 44.28, -46.686]
  Call Extruder(148.23578)
  MoveL 295 to (-27.53, 35.73, 22.23) mm, rotated rx 180 ry 0 rz 180 deg; joints [-35.317, -19.484, 80.876, 55.949, 44.246, -46.668]
  MoveL 296 to (-27.53, 35.73, 22.23) mm, rotated rx 180 ry 0 rz 180 deg; joints [-35.317, -19.484, 80.876, 55.949, 44.246, -46.668]
  Call Extruder(148.51252)
  MoveL 297 to (-27.28, 35.68, 22.22) mm, rotated rx 180 ry 0 rz 180 deg; joints [-35.278, -19.461, 80.862, 55.917, 44.213, -46.65]
  MoveL 298 to (-27.28, 35.68, 22.22) mm, rotated rx 180 ry 0 rz 180 deg; joints [-35.278, -19.461, 80.862, 55.917, 44.213, -46.65]
  Call Extruder(148.72072)
  MoveL 299 to (-27.09, 35.65, 22.22) mm, rotated rx 180 ry 0 rz 180 deg; joints [-35.248, -19.444, 80.852, 55.893, 44.187, -46.637]
  MoveL 300 to (-27.09, 35.65, 22.22) mm, rotated rx 180 ry 0 rz 180 deg; joints [-35.248, -19.444, 80.852, 55.893, 44.187, -46.637]
  Call Extruder(148.95842)
  MoveL 301 to (-26.87, 35.61, 22.22) mm, rotated rx -180 ry 0 rz -180 deg; joints [-35.215, -19.425, 80.84, 55.867, 44.159, -46.622]
  MoveL 302 to (-26.87, 35.61, 22.22) mm, rotated rx -180 ry 0 rz -180 deg; joints [-35.215, -19.425, 80.84, 55.867, 44.159, -46.622]
  Call Extruder(149.29181)
  MoveL 303 to (-26.57, 35.56, 22.22) mm, rotated rx -180 ry 0 rz 180 deg; joints [-35.168, -19.397, 80.823, 55.83, 44.119, -46.602]
  MoveL 304 to (-26.57, 35.56, 22.22) mm, rotated rx -180 ry 0 rz 180 deg; joints [-35.168, -19.397, 80.823, 55.83, 44.119, -46.602]
  Call Extruder(149.62348)
  MoveL 305 to (-26.26, 35.51, 22.23) mm, rotated rx 180 ry 0 rz 180 deg; joints [-35.122, -19.368, 80.805, 55.794, 44.079, -46.583]
  MoveL 306 to (-26.26, 35.51, 22.23) mm, rotated rx 180 ry 0 rz 180 deg; joints [-35.122, -19.368, 80.805, 55.794, 44.079, -46.583]
  Call Extruder(149.95342)
  MoveL 307 to (-25.96, 35.47, 22.22) mm, rotated rx 180 ry 0 rz 180 deg; joints [-35.075, -19.34, 80.788, 55.757, 44.039, -46.563]
  MoveL 308 to (-25.96, 35.47, 22.22) mm, rotated rx 180 ry 0 rz 180 deg; joints [-35.075, -19.34, 80.788, 55.757, 44.039, -46.563]
  Call Extruder(150.28165)
  MoveL 309 to (-25.65, 35.42, 22.22) mm, rotated rx 180 ry 0 rz 180 deg; joints [-35.029, -19.312, 80.771, 55.721, 43.999, -46.543]
  MoveL 310 to (-25.65, 35.42, 22.22) mm, rotated rx 180 ry 0 rz 180 deg; joints [-35.029, -19.312, 80.771, 55.721, 43.999, -46.543]
  Call Extruder(150.60817)
  MoveL 311 to (-25.34, 35.37, 22.22) mm, rotated rx 180 ry 0 rz 180 deg; joints [-34.983, -19.283, 80.753, 55.685, 43.96, -46.523]
  MoveL 312 to (-25.34, 35.37, 22.22) mm, rotated rx 180 ry 0 rz 180 deg; joints [-34.983, -19.283, 80.753, 55.685, 43.96, -46.523]
  Call Extruder(150.97524)
  MoveL 313 to (-25, 35.32, 22.22) mm, rotated rx -180 ry 0 rz 180 deg; joints [-34.932, -19.251, 80.733, 55.645, 43.916, -46.502]
  MoveL 314 to (-25, 35.32, 22.22) mm, rotated rx -180 ry 0 rz 180 deg; joints [-34.932, -19.251, 80.733, 55.645, 43.916, -46.502]
  Call Extruder(151.38268)
  MoveL 315 to (-24.61, 35.27, 22.22) mm, rotated rx 180 ry 0 rz 180 deg; joints [-34.877, -19.213, 80.71, 55.602, 43.867, -46.479]
  MoveL 316 to (-24.61, 35.27, 22.22) mm, rotated rx 180 ry 0 rz 180 deg; joints [-34.877, -19.213, 80.71, 55.602, 43.867, -46.479]
  Call Extruder(151.78808)
  MoveL 317 to (-24.22, 35.23, 22.22) mm, rotated rx 180 ry 0 rz 180 deg; joints [-34.821, -19.176, 80.687, 55.559, 43.819, -46.456]
  MoveL 318 to (-24.22, 35.23, 22.22) mm, rotated rx 180 ry 0 rz 180 deg; joints [-34.821, -19.176, 80.687, 55.559, 43.819, -46.456]
  Call Extruder(152.19142)
  MoveL 319 to (-23.84, 35.18, 22.22) mm, rotated rx 180 ry 0 rz 180 deg; joints [-34.766, -19.139, 80.664, 55.517, 43.771, -46.433]
  MoveL 320 to (-23.84, 35.18, 22.22) mm, rotated rx 180 ry 0 rz 180 deg; joints [-34.766, -19.139, 80.664, 55.517, 43.771, -46.433]
  Call Extruder(152.59271)
  MoveL 321 to (-23.45, 35.14, 22.22) mm, rotated rx 180 ry 0 rz 180 deg; joints [-34.711, -19.101, 80.641, 55.474, 43.723, -46.411]
  MoveL 322 to (-23.45, 35.14, 22.22) mm, rotated rx 180 ry 0 rz 180 deg; joints [-34.711, -19.101, 80.641, 55.474, 43.723, -46.411]
  Call Extruder(153.19759)
  MoveL 323 to (-22.86, 35.09, 22.23) mm, rotated rx -180 ry 0 rz 180 deg; joints [-34.631, -19.043, 80.605, 55.414, 43.653, -46.38]
  MoveL 324 to (-22.86, 35.09, 22.23) mm, rotated rx -180 ry 0 rz 180 deg; joints [-34.631, -19.043, 80.605, 55.414, 43.653, -46.38]
  Call Extruder(153.79932)
  MoveL 325 to (-22.27, 35.05, 22.22) mm, rotated rx 180 ry 0 rz 180 deg; joints [-34.552, -18.984, 80.568, 55.354, 43.583, -46.349]
  MoveL 326 to (-22.27, 35.05, 22.22) mm, rotated rx 180 ry 0 rz 180 deg; joints [-34.552, -18.984, 80.568, 55.354, 43.583, -46.349]
  Call Extruder(154.39790)
  MoveL 327 to (-21.68, 35, 22.22) mm, rotated rx 180 ry 0 rz 180 deg; joints [-34.473, -18.926, 80.532, 55.294, 43.513, -46.318]
  MoveL 328 to (-21.68, 35, 22.22) mm, rotated rx 180 ry 0 rz 180 deg; joints [-34.473, -18.926, 80.532, 55.294, 43.513, -46.318]
  Call Extruder(155.56967)
  MoveL 329 to (-20.52, 34.95, 22.22) mm, rotated rx 180 ry 0 rz 180 deg; joints [-34.326, -18.806, 80.457, 55.185, 43.381, -46.265]
  MoveL 330 to (-20.52, 34.95, 22.22) mm, rotated rx 180 ry 0 rz 180 deg; joints [-34.326, -18.806, 80.457, 55.185, 43.381, -46.265]
  Call Extruder(157.02754)
  MoveL 331 to (-19.06, 34.91, 22.22) mm, rotated rx 180 ry 0 rz 180 deg; joints [-34.146, -18.655, 80.363, 55.053, 43.219, -46.2]
  Call Extruder(395.62063)
  MoveL 332 to (219.06, 34.91, 22.22) mm, rotated rx 180 ry 0 rz 180 deg; joints [-18.248, 14.754, 48.244, 35.988, 32.201, -31.572]
  Call Extruder(396.49572)
  MoveL 333 to (219.94, 34.93, 22.22) mm, rotated rx 180 ry 0 rz 180 deg; joints [-18.218, 14.928, 48.02, 35.893, 32.226, -31.475]
  MoveL 334 to (219.94, 34.93, 22.22) mm, rotated rx 180 ry 0 rz 180 deg; joints [-18.218, 14.928, 48.02, 35.893, 32.226, -31.475]
  Call Extruder(397.66749)
  MoveL 335 to (221.1, 34.97, 22.23) mm, rotated rx -180 ry 0 rz 180 deg; joints [-18.181, 15.162, 47.717, 35.769, 32.263, -31.348]
  MoveL 336 to (221.1, 34.97, 22.23) mm, rotated rx -180 ry 0 rz 180 deg; joints [-18.181, 15.162, 47.717, 35.769, 32.263, -31.348]
  Call Extruder(398.55557)
  MoveL 337 to (221.97, 35.02, 22.23) mm, rotated rx 180 ry 0 rz -180 deg; joints [-18.154, 15.34, 47.485, 35.676, 32.292, -31.254]
  MoveL 338 to (221.97, 35.02, 22.23) mm, rotated rx 180 ry 0 rz -180 deg; joints [-18.154, 15.34, 47.485, 35.676, 32.292, -31.254]
  Call Extruder(399.15730)
  MoveL 339 to (222.56, 35.07, 22.22) mm, rotated rx 180 ry 0 rz 180 deg; joints [-18.138, 15.461, 47.327, 35.616, 32.314, -31.192]
  MoveL 340 to (222.56, 35.07, 22.22) mm, rotated rx 180 ry 0 rz 180 deg; joints [-18.138, 15.461, 47.327, 35.616, 32.314, -31.192]
  Call Extruder(399.76217)
  MoveL 341 to (223.15, 35.11, 22.23) mm, rotated rx 180 ry 0 rz 180 deg; joints [-18.121, 15.583, 47.168, 35.556, 32.336, -31.129]
  MoveL 342 to (223.15, 35.11, 22.23) mm, rotated rx 180 ry 0 rz 180 deg; joints [-18.121, 15.583, 47.168, 35.556, 32.336, -31.129]
  Call Extruder(400.26672)
  MoveL 343 to (223.64, 35.16, 22.23) mm, rotated rx 180 ry 0 rz 180 deg; joints [-18.109, 15.685, 47.035, 35.507, 32.355, -31.078]
  MoveL 344 to (223.64, 35.16, 22.23) mm, rotated rx 180 ry 0 rz 180 deg; joints [-18.109, 15.685, 47.035, 35.507, 32.355, -31.078]
  Call Extruder(400.67007)
  MoveL 345 to (224.03, 35.21, 22.22) mm, rotated rx 180 ry 0 rz -180 deg; joints [-18.1, 15.766, 46.928, 35.47, 32.371, -31.038]
  MoveL 346 to (224.03, 35.21, 22.22) mm, rotated rx 180 ry 0 rz -180 deg; joints [-18.1, 15.766, 46.928, 35.47, 32.371, -31.038]
  Call Extruder(401.07546)
  MoveL 347 to (224.42, 35.25, 22.23) mm, rotated rx 180 ry 0 rz 180 deg; joints [-18.091, 15.848, 46.821, 35.432, 32.387, -30.999]
  MoveL 348 to (224.42, 35.25, 22.23) mm, rotated rx 180 ry 0 rz 180 deg; joints [-18.091, 15.848, 46.821, 35.432, 32.387, -30.999]
  Call Extruder(401.48291)
  MoveL 349 to (224.8, 35.3, 22.22) mm, rotated rx 180 ry 0 rz 180 deg; joints [-18.082, 15.93, 46.713, 35.394, 32.404, -30.959]
  MoveL 350 to (224.8, 35.3, 22.22) mm, rotated rx 180 ry 0 rz 180 deg; joints [-18.082, 15.93, 46.713, 35.394, 32.404, -30.959]
  Call Extruder(401.89240)
  MoveL 351 to (225.19, 35.34, 22.23) mm, rotated rx 180 ry 0 rz 180 deg; joints [-18.073, 16.012, 46.605, 35.356, 32.42, -30.919]
  MoveL 352 to (225.19, 35.34, 22.23) mm, rotated rx 180 ry 0 rz 180 deg; joints [-18.073, 16.012, 46.605, 35.356, 32.42, -30.919]
  Call Extruder(402.21894)
  MoveL 353 to (225.5, 35.39, 22.23) mm, rotated rx -180 ry 0 rz 180 deg; joints [-18.068, 16.078, 46.518, 35.328, 32.434, -30.889]
  MoveL 354 to (225.5, 35.39, 22.23) mm, rotated rx -180 ry 0 rz 180 deg; joints [-18.068, 16.078, 46.518, 35.328, 32.434, -30.889]
  Call Extruder(402.54719)
  MoveL 355 to (225.8, 35.44, 22.22) mm, rotated rx 180 ry 0 rz 180 deg; joints [-18.062, 16.144, 46.431, 35.3, 32.448, -30.858]
  MoveL 356 to (225.8, 35.44, 22.22) mm, rotated rx 180 ry 0 rz 180 deg; joints [-18.062, 16.144, 46.431, 35.3, 32.448, -30.858]
  Call Extruder(402.87716)
  MoveL 357 to (226.11, 35.49, 22.22) mm, rotated rx 180 ry 0 rz 180 deg; joints [-18.056, 16.209, 46.345, 35.272, 32.463, -30.828]
  MoveL 358 to (226.11, 35.49, 22.22) mm, rotated rx 180 ry 0 rz 180 deg; joints [-18.056, 16.209, 46.345, 35.272, 32.463, -30.828]
  Call Extruder(403.20885)
  MoveL 359 to (226.41, 35.54, 22.23) mm, rotated rx 180 ry 0 rz 180 deg; joints [-18.051, 16.276, 46.257, 35.244, 32.477, -30.798]
  MoveL 360 to (226.41, 35.54, 22.23) mm, rotated rx 180 ry 0 rz 180 deg; joints [-18.051, 16.276, 46.257, 35.244, 32.477, -30.798]
  Call Extruder(403.54226)
  MoveL 361 to (226.72, 35.59, 22.22) mm, rotated rx -180 ry 0 rz 180 deg; joints [-18.045, 16.342, 46.169, 35.215, 32.492, -30.767]
  MoveL 362 to (226.72, 35.59, 22.22) mm, rotated rx -180 ry 0 rz 180 deg; joints [-18.045, 16.342, 46.169, 35.215, 32.492, -30.767]
  Call Extruder(403.87738)
  MoveL 363 to (227.03, 35.64, 22.22) mm, rotated rx 180 ry 0 rz -180 deg; joints [-18.039, 16.408, 46.082, 35.187, 32.506, -30.737]
  MoveL 364 to (227.03, 35.64, 22.22) mm, rotated rx 180 ry 0 rz -180 deg; joints [-18.039, 16.408, 46.082, 35.187, 32.506, -30.737]
  Call Extruder(404.15384)
  MoveL 365 to (227.28, 35.68, 22.22) mm, rotated rx -180 ry 0 rz 180 deg; joints [-18.036, 16.463, 46.009, 35.165, 32.519, -30.713]
  MoveL 366 to (227.28, 35.68, 22.22) mm, rotated rx -180 ry 0 rz 180 deg; joints [-18.036, 16.463, 46.009, 35.165, 32.519, -30.713]
  Call Extruder(404.43174)
  MoveL 367 to (227.52, 35.73, 22.22) mm, rotated rx 180 ry 0 rz 180 deg; joints [-18.033, 16.518, 45.936, 35.144, 32.532, -30.689]
  MoveL 368 to (227.52, 35.73, 22.22) mm, rotated rx 180 ry 0 rz 180 deg; joints [-18.033, 16.518, 45.936, 35.144, 32.532, -30.689]
  Call Extruder(404.71108)
  MoveL 369 to (227.77, 35.78, 22.22) mm, rotated rx -180 ry 0 rz 180 deg; joints [-18.029, 16.573, 45.863, 35.122, 32.545, -30.665]
  MoveL 370 to (227.77, 35.78, 22.22) mm, rotated rx -180 ry 0 rz 180 deg; joints [-18.029, 16.573, 45.863, 35.122, 32.545, -30.665]
  Call Extruder(404.99186)
  MoveL 371 to (228.02, 35.83, 22.22) mm, rotated rx -180 ry 0 rz 180 deg; joints [-18.026, 16.628, 45.789, 35.1, 32.558, -30.641]
  MoveL 372 to (228.02, 35.83, 22.22) mm, rotated rx -180 ry 0 rz 180 deg; joints [-18.026, 16.628, 45.789, 35.1, 32.558, -30.641]
  Call Extruder(405.27408)
  MoveL 373 to (228.27, 35.88, 22.23) mm, rotated rx -180 ry 0 rz 180 deg; joints [-18.022, 16.684, 45.716, 35.078, 32.571, -30.617]
  MoveL 374 to (228.27, 35.88, 22.23) mm, rotated rx -180 ry 0 rz 180 deg; joints [-18.022, 16.684, 45.716, 35.078, 32.571, -30.617]
  Call Extruder(405.55775)
  MoveL 375 to (228.52, 35.93, 22.23) mm, rotated rx 180 ry 0 rz 180 deg; joints [-18.019, 16.739, 45.642, 35.056, 32.585, -30.592]
  MoveL 376 to (228.52, 35.93, 22.23) mm, rotated rx 180 ry 0 rz 180 deg; joints [-18.019, 16.739, 45.642, 35.056, 32.585, -30.592]
  Call Extruder(405.84286)
  MoveL 377 to (228.77, 35.98, 22.22) mm, rotated rx 180 ry 0 rz 180 deg; joints [-18.015, 16.794, 45.569, 35.034, 32.598, -30.568]
  MoveL 378 to (228.77, 35.98, 22.22) mm, rotated rx 180 ry 0 rz 180 deg; joints [-18.015, 16.794, 45.569, 35.034, 32.598, -30.568]
  Call Extruder(406.07863)
  MoveL 379 to (228.97, 36.03, 22.22) mm, rotated rx 180 ry 0 rz 180 deg; joints [-18.013, 16.84, 45.508, 35.016, 32.609, -30.549]
  MoveL 380 to (228.97, 36.03, 22.22) mm, rotated rx 180 ry 0 rz 180 deg; joints [-18.013, 16.84, 45.508, 35.016, 32.609, -30.549]
  Call Extruder(406.31548)
  MoveL 381 to (229.18, 36.07, 22.23) mm, rotated rx -180 ry 0 rz 180 deg; joints [-18.01, 16.886, 45.446, 34.999, 32.621, -30.529]
  MoveL 382 to (229.18, 36.07, 22.23) mm, rotated rx -180 ry 0 rz 180 deg; joints [-18.01, 16.886, 45.446, 34.999, 32.621, -30.529]
  Call Extruder(406.55339)
  MoveL 383 to (229.38, 36.12, 22.22) mm, rotated rx -180 ry 0 rz 180 deg; joints [-18.008, 16.932, 45.385, 34.981, 32.632, -30.51]
  MoveL 384 to (229.38, 36.12, 22.22) mm, rotated rx -180 ry 0 rz 180 deg; joints [-18.008, 16.932, 45.385, 34.981, 32.632, -30.51]
  Call Extruder(406.79238)
  MoveL 385 to (229.59, 36.16, 22.23) mm, rotated rx 180 ry 0 rz 180 deg; joints [-18.006, 16.978, 45.324, 34.964, 32.643, -30.49]
  MoveL 386 to (229.59, 36.16, 22.23) mm, rotated rx 180 ry 0 rz 180 deg; joints [-18.006, 16.978, 45.324, 34.964, 32.643, -30.49]
  Call Extruder(407.04637)
  MoveL 387 to (229.8, 36.22, 22.22) mm, rotated rx -180 ry 0 rz 180 deg; joints [-18.004, 17.027, 45.258, 34.947, 32.656, -30.47]
  MoveL 388 to (229.8, 36.22, 22.22) mm, rotated rx -180 ry 0 rz 180 deg; joints [-18.004, 17.027, 45.258, 34.947, 32.656, -30.47]
  Call Extruder(407.31597)
  MoveL 389 to (230.02, 36.28, 22.22) mm, rotated rx -180 ry 0 rz 180 deg; joints [-18.004, 17.079, 45.189, 34.93, 32.67, -30.451]
  MoveL 390 to (230.02, 36.28, 22.22) mm, rotated rx -180 ry 0 rz 180 deg; joints [-18.004, 17.079, 45.189, 34.93, 32.67, -30.451]
  Call Extruder(407.58690)
  MoveL 391 to (230.25, 36.35, 22.23) mm, rotated rx -180 ry 0 rz 180 deg; joints [-18.003, 17.131, 45.119, 34.914, 32.684, -30.432]
  MoveL 392 to (230.25, 36.35, 22.23) mm, rotated rx -180 ry 0 rz 180 deg; joints [-18.003, 17.131, 45.119, 34.914, 32.684, -30.432]
  Call Extruder(407.85917)
  MoveL 393 to (230.47, 36.42, 22.22) mm, rotated rx 180 ry 0 rz -180 deg; joints [-18.003, 17.183, 45.05, 34.897, 32.699, -30.412]
  MoveL 394 to (230.47, 36.42, 22.22) mm, rotated rx 180 ry 0 rz -180 deg; joints [-18.003, 17.183, 45.05, 34.897, 32.699, -30.412]
  Call Extruder(408.13278)
  MoveL 395 to (230.7, 36.49, 22.23) mm, rotated rx -180 ry 0 rz 180 deg; joints [-18.002, 17.235, 44.98, 34.88, 32.713, -30.393]
  MoveL 396 to (230.7, 36.49, 22.23) mm, rotated rx -180 ry 0 rz 180 deg; joints [-18.002, 17.235, 44.98, 34.88, 32.713, -30.393]
  Call Extruder(408.36597)
  MoveL 397 to (230.88, 36.55, 22.22) mm, rotated rx -180 ry 0 rz 180 deg; joints [-18.002, 17.279, 44.92, 34.867, 32.725, -30.377]
  MoveL 398 to (230.88, 36.55, 22.22) mm, rotated rx -180 ry 0 rz 180 deg; joints [-18.002, 17.279, 44.92, 34.867, 32.725, -30.377]
  Call Extruder(408.60021)
  MoveL 399 to (231.07, 36.61, 22.22) mm, rotated rx 180 ry 0 rz 180 deg; joints [-18.002, 17.323, 44.861, 34.853, 32.738, -30.361]
  MoveL 400 to (231.07, 36.61, 22.22) mm, rotated rx 180 ry 0 rz 180 deg; joints [-18.002, 17.323, 44.861, 34.853, 32.738, -30.361]
  Call Extruder(408.83551)
  MoveL 401 to (231.26, 36.67, 22.22) mm, rotated rx -180 ry 0 rz 180 deg; joints [-18.002, 17.368, 44.801, 34.84, 32.75, -30.345]
  MoveL 402 to (231.26, 36.67, 22.22) mm, rotated rx -180 ry 0 rz 180 deg; joints [-18.002, 17.368, 44.801, 34.84, 32.75, -30.345]
  Call Extruder(409.07185)
  MoveL 403 to (231.45, 36.73, 22.23) mm, rotated rx 180 ry 0 rz -180 deg; joints [-18.002, 17.412, 44.741, 34.826, 32.763, -30.328]
  MoveL 404 to (231.45, 36.73, 22.23) mm, rotated rx 180 ry 0 rz -180 deg; joints [-18.002, 17.412, 44.741, 34.826, 32.763, -30.328]
  Call Extruder(409.30925)
  MoveL 405 to (231.64, 36.79, 22.22) mm, rotated rx -180 ry 0 rz 180 deg; joints [-18.002, 17.457, 44.682, 34.812, 32.776, -30.312]
  MoveL 406 to (231.64, 36.79, 22.22) mm, rotated rx -180 ry 0 rz 180 deg; joints [-18.002, 17.457, 44.682, 34.812, 32.776, -30.312]
  Call Extruder(409.68944)
  MoveL 407 to (231.93, 36.91, 22.23) mm, rotated rx 180 ry 0 rz 180 deg; joints [-18.005, 17.527, 44.586, 34.795, 32.797, -30.29]
  MoveL 408 to (231.93, 36.91, 22.23) mm, rotated rx 180 ry 0 rz 180 deg; joints [-18.005, 17.527, 44.586, 34.795, 32.797, -30.29]
  Call Extruder(410.07143)
  MoveL 409 to (232.22, 37.04, 22.22) mm, rotated rx -180 ry 0 rz 180 deg; joints [-18.008, 17.598, 44.49, 34.778, 32.819, -30.268]
  MoveL 410 to (232.22, 37.04, 22.22) mm, rotated rx -180 ry 0 rz 180 deg; joints [-18.008, 17.598, 44.49, 34.778, 32.819, -30.268]
  Call Extruder(410.42789)
  MoveL 411 to (232.49, 37.15, 22.22) mm, rotated rx -180 ry 0 rz -180 deg; joints [-18.011, 17.664, 44.401, 34.762, 32.839, -30.247]
  MoveL 412 to (232.49, 37.15, 22.22) mm, rotated rx -180 ry 0 rz -180 deg; joints [-18.011, 17.664, 44.401, 34.762, 32.839, -30.247]
  Call Extruder(410.75854)
  MoveL 413 to (232.74, 37.26, 22.22) mm, rotated rx 180 ry 0 rz 180 deg; joints [-18.013, 17.726, 44.319, 34.747, 32.858, -30.228]
  MoveL 414 to (232.74, 37.26, 22.22) mm, rotated rx 180 ry 0 rz 180 deg; joints [-18.013, 17.726, 44.319, 34.747, 32.858, -30.228]
  Call Extruder(411.09062)
  MoveL 415 to (232.99, 37.36, 22.22) mm, rotated rx -180 ry 0 rz 180 deg; joints [-18.016, 17.787, 44.236, 34.733, 32.878, -30.209]
  MoveL 416 to (232.99, 37.36, 22.22) mm, rotated rx -180 ry 0 rz 180 deg; joints [-18.016, 17.787, 44.236, 34.733, 32.878, -30.209]
  Call Extruder(411.52249)
  MoveL 417 to (233.29, 37.54, 22.22) mm, rotated rx 180 ry 0 rz 180 deg; joints [-18.024, 17.865, 44.13, 34.721, 32.905, -30.191]
  MoveL 418 to (233.29, 37.54, 22.22) mm, rotated rx 180 ry 0 rz 180 deg; joints [-18.024, 17.865, 44.13, 34.721, 32.905, -30.191]
  Call Extruder(411.95620)
  MoveL 419 to (233.6, 37.71, 22.23) mm, rotated rx 180 ry 0 rz 180 deg; joints [-18.033, 17.943, 44.024, 34.71, 32.932, -30.173]
  MoveL 420 to (233.6, 37.71, 22.23) mm, rotated rx 180 ry 0 rz 180 deg; joints [-18.033, 17.943, 44.024, 34.71, 32.932, -30.173]
  Call Extruder(412.39175)
  MoveL 421 to (233.9, 37.89, 22.23) mm, rotated rx 180 ry 0 rz 180 deg; joints [-18.041, 18.022, 43.917, 34.699, 32.959, -30.155]
  MoveL 422 to (233.9, 37.89, 22.23) mm, rotated rx 180 ry 0 rz 180 deg; joints [-18.041, 18.022, 43.917, 34.699, 32.959, -30.155]
  Call Extruder(412.82915)
  MoveL 423 to (234.21, 38.07, 22.23) mm, rotated rx -180 ry 0 rz 180 deg; joints [-18.049, 18.101, 43.81, 34.687, 32.986, -30.137]
  MoveL 424 to (234.21, 38.07, 22.23) mm, rotated rx -180 ry 0 rz 180 deg; joints [-18.049, 18.101, 43.81, 34.687, 32.986, -30.137]
  Call Extruder(413.20589)
  MoveL 425 to (234.45, 38.24, 22.22) mm, rotated rx 180 ry 0 rz 180 deg; joints [-18.06, 18.167, 43.72, 34.683, 33.011, -30.125]
  MoveL 426 to (234.45, 38.24, 22.22) mm, rotated rx 180 ry 0 rz 180 deg; joints [-18.06, 18.167, 43.72, 34.683, 33.011, -30.125]
  Call Extruder(413.90582)
  MoveL 427 to (234.9, 38.57, 22.22) mm, rotated rx 180 ry 0 rz 180 deg; joints [-18.079, 18.289, 43.554, 34.675, 33.057, -30.105]
  MoveL 428 to (234.9, 38.57, 22.22) mm, rotated rx 180 ry 0 rz 180 deg; joints [-18.079, 18.289, 43.554, 34.675, 33.057, -30.105]
  Call Extruder(414.60855)
  MoveL 429 to (235.35, 38.9, 22.23) mm, rotated rx 180 ry 0 rz 180 deg; joints [-18.099, 18.412, 43.386, 34.666, 33.104, -30.084]
  Call Extruder(416.34741)
  MoveL 430 to (236.39, 39.81, 22.22) mm, rotated rx 180 ry 0 rz -180 deg; joints [-18.16, 18.708, 42.98, 34.669, 33.225, -30.052]
  Call Extruder(418.08626)
  MoveL 431 to (237.3, 40.85, 22.22) mm, rotated rx -180 ry 0 rz 180 deg; joints [-18.24, 18.988, 42.595, 34.702, 33.351, -30.047]
  Call Extruder(418.43762)
  MoveL 432 to (237.47, 41.07, 22.22) mm, rotated rx -180 ry 0 rz 180 deg; joints [-18.258, 19.042, 42.521, 34.714, 33.377, -30.05]
  MoveL 433 to (237.47, 41.07, 22.22) mm, rotated rx -180 ry 0 rz 180 deg; joints [-18.258, 19.042, 42.521, 34.714, 33.377, -30.05]
  Call Extruder(419.13755)
  MoveL 434 to (237.8, 41.52, 22.22) mm, rotated rx -180 ry 0 rz 180 deg; joints [-18.295, 19.149, 42.372, 34.736, 33.429, -30.056]
  MoveL 435 to (237.8, 41.52, 22.22) mm, rotated rx -180 ry 0 rz 180 deg; joints [-18.295, 19.149, 42.372, 34.736, 33.429, -30.056]
  Call Extruder(419.83467)
  MoveL 436 to (238.12, 41.97, 22.22) mm, rotated rx 180 ry 0 rz 180 deg; joints [-18.332, 19.258, 42.222, 34.758, 33.482, -30.061]
  MoveL 437 to (238.12, 41.97, 22.22) mm, rotated rx 180 ry 0 rz 180 deg; joints [-18.332, 19.258, 42.222, 34.758, 33.482, -30.061]
  Call Extruder(420.08158)
  MoveL 438 to (238.22, 42.15, 22.22) mm, rotated rx 180 ry 0 rz 180 deg; joints [-18.346, 19.293, 42.173, 34.769, 33.501, -30.067]
  MoveL 439 to (238.22, 42.15, 22.22) mm, rotated rx 180 ry 0 rz 180 deg; joints [-18.346, 19.293, 42.173, 34.769, 33.501, -30.067]
  Call Extruder(420.51713)
  MoveL 440 to (238.4, 42.45, 22.23) mm, rotated rx 180 ry 0 rz -180 deg; joints [-18.373, 19.356, 42.086, 34.79, 33.534, -30.076]
  MoveL 441 to (238.4, 42.45, 22.23) mm, rotated rx 180 ry 0 rz -180 deg; joints [-18.373, 19.356, 42.086, 34.79, 33.534, -30.076]
  Call Extruder(420.95084)
  MoveL 442 to (238.57, 42.75, 22.22) mm, rotated rx 180 ry 0 rz -180 deg; joints [-18.399, 19.419, 41.999, 34.81, 33.567, -30.085]
  MoveL 443 to (238.57, 42.75, 22.22) mm, rotated rx 180 ry 0 rz -180 deg; joints [-18.399, 19.419, 41.999, 34.81, 33.567, -30.085]
  Call Extruder(421.38271)
  MoveL 444 to (238.75, 43.06, 22.22) mm, rotated rx 180 ry 0 rz 180 deg; joints [-18.425, 19.482, 41.911, 34.83, 33.6, -30.094]
  MoveL 445 to (238.75, 43.06, 22.22) mm, rotated rx 180 ry 0 rz 180 deg; joints [-18.425, 19.482, 41.911, 34.83, 33.6, -30.094]
  Call Extruder(421.76312)
  MoveL 446 to (238.89, 43.34, 22.23) mm, rotated rx 180 ry 0 rz 180 deg; joints [-18.45, 19.536, 41.836, 34.85, 33.63, -30.104]
  MoveL 447 to (238.89, 43.34, 22.23) mm, rotated rx 180 ry 0 rz 180 deg; joints [-18.45, 19.536, 41.836, 34.85, 33.63, -30.104]
  Call Extruder(422.09380)
  MoveL 448 to (239, 43.58, 22.22) mm, rotated rx 180 ry 0 rz 180 deg; joints [-18.472, 19.579, 41.776, 34.871, 33.655, -30.116]
  MoveL 449 to (239, 43.58, 22.22) mm, rotated rx 180 ry 0 rz 180 deg; joints [-18.472, 19.579, 41.776, 34.871, 33.655, -30.116]
  Call Extruder(422.42305)
  MoveL 450 to (239.11, 43.83, 22.23) mm, rotated rx 180 ry 0 rz 180 deg; joints [-18.495, 19.623, 41.715, 34.892, 33.681, -30.128]
  MoveL 451 to (239.11, 43.83, 22.23) mm, rotated rx 180 ry 0 rz 180 deg; joints [-18.495, 19.623, 41.715, 34.892, 33.681, -30.128]
  Call Extruder(422.80503)
  MoveL 452 to (239.23, 44.13, 22.23) mm, rotated rx 180 ry 0 rz 180 deg; joints [-18.522, 19.673, 41.645, 34.917, 33.71, -30.142]
  MoveL 453 to (239.23, 44.13, 22.23) mm, rotated rx 180 ry 0 rz 180 deg; joints [-18.522, 19.673, 41.645, 34.917, 33.71, -30.142]
  Call Extruder(423.18522)
  MoveL 454 to (239.35, 44.42, 22.22) mm, rotated rx 180 ry 0 rz 180 deg; joints [-18.549, 19.723, 41.575, 34.941, 33.74, -30.157]
  MoveL 455 to (239.35, 44.42, 22.22) mm, rotated rx 180 ry 0 rz 180 deg; joints [-18.549, 19.723, 41.575, 34.941, 33.74, -30.157]
  Call Extruder(423.49290)
  MoveL 456 to (239.44, 44.66, 22.22) mm, rotated rx 180 ry 0 rz 180 deg; joints [-18.571, 19.763, 41.52, 34.963, 33.764, -30.169]
  MoveL 457 to (239.44, 44.66, 22.22) mm, rotated rx 180 ry 0 rz 180 deg; joints [-18.571, 19.763, 41.52, 34.963, 33.764, -30.169]
  Call Extruder(423.72925)
  MoveL 458 to (239.5, 44.85, 22.23) mm, rotated rx -180 ry 0 rz 180 deg; joints [-18.589, 19.792, 41.479, 34.981, 33.782, -30.181]
  MoveL 459 to (239.5, 44.85, 22.23) mm, rotated rx -180 ry 0 rz 180 deg; joints [-18.589, 19.792, 41.479, 34.981, 33.782, -30.181]
  Call Extruder(423.96455)
  MoveL 460 to (239.56, 45.03, 22.23) mm, rotated rx -180 ry 0 rz 180 deg; joints [-18.607, 19.821, 41.439, 34.998, 33.801, -30.192]
  MoveL 461 to (239.56, 45.03, 22.23) mm, rotated rx -180 ry 0 rz 180 deg; joints [-18.607, 19.821, 41.439, 34.998, 33.801, -30.192]
  Call Extruder(424.19880)
  MoveL 462 to (239.62, 45.22, 22.22) mm, rotated rx 180 ry 0 rz 180 deg; joints [-18.625, 19.849, 41.399, 35.016, 33.819, -30.203]
  MoveL 463 to (239.62, 45.22, 22.22) mm, rotated rx 180 ry 0 rz 180 deg; joints [-18.625, 19.849, 41.399, 35.016, 33.819, -30.203]
  Call Extruder(424.43200)
  MoveL 464 to (239.68, 45.41, 22.22) mm, rotated rx -180 ry 0 rz 180 deg; joints [-18.642, 19.878, 41.359, 35.034, 33.837, -30.214]
  MoveL 465 to (239.68, 45.41, 22.22) mm, rotated rx -180 ry 0 rz 180 deg; joints [-18.642, 19.878, 41.359, 35.034, 33.837, -30.214]
  Call Extruder(424.68486)
  MoveL 466 to (239.75, 45.62, 22.22) mm, rotated rx -180 ry 0 rz 180 deg; joints [-18.662, 19.909, 41.315, 35.054, 33.857, -30.227]
  MoveL 467 to (239.75, 45.62, 22.22) mm, rotated rx -180 ry 0 rz 180 deg; joints [-18.662, 19.909, 41.315, 35.054, 33.857, -30.227]
  Call Extruder(424.95712)
  MoveL 468 to (239.82, 45.84, 22.23) mm, rotated rx -180 ry 0 rz 180 deg; joints [-18.683, 19.943, 41.268, 35.076, 33.879, -30.24]
  MoveL 469 to (239.82, 45.84, 22.23) mm, rotated rx -180 ry 0 rz 180 deg; joints [-18.683, 19.943, 41.268, 35.076, 33.879, -30.24]
  Call Extruder(425.22805)
  MoveL 470 to (239.88, 46.06, 22.22) mm, rotated rx -180 ry 0 rz 180 deg; joints [-18.705, 19.976, 41.222, 35.097, 33.901, -30.254]
  MoveL 471 to (239.88, 46.06, 22.22) mm, rotated rx -180 ry 0 rz 180 deg; joints [-18.705, 19.976, 41.222, 35.097, 33.901, -30.254]
  Call Extruder(425.49763)
  MoveL 472 to (239.95, 46.29, 22.23) mm, rotated rx -180 ry 0 rz 180 deg; joints [-18.726, 20.009, 41.175, 35.119, 33.922, -30.268]
  MoveL 473 to (239.95, 46.29, 22.23) mm, rotated rx -180 ry 0 rz 180 deg; joints [-18.726, 20.009, 41.175, 35.119, 33.922, -30.268]
  Call Extruder(425.76589)
  MoveL 474 to (240.02, 46.51, 22.22) mm, rotated rx 180 ry 0 rz 180 deg; joints [-18.747, 20.043, 41.128, 35.14, 33.944, -30.281]
  MoveL 475 to (240.02, 46.51, 22.22) mm, rotated rx 180 ry 0 rz 180 deg; joints [-18.747, 20.043, 41.128, 35.14, 33.944, -30.281]
  Call Extruder(426.00483)
  MoveL 476 to (240.06, 46.72, 22.22) mm, rotated rx 180 ry 0 rz 180 deg; joints [-18.767, 20.069, 41.091, 35.162, 33.963, -30.296]
  MoveL 477 to (240.06, 46.72, 22.22) mm, rotated rx 180 ry 0 rz 180 deg; joints [-18.767, 20.069, 41.091, 35.162, 33.963, -30.296]
  Call Extruder(426.24270)
  MoveL 478 to (240.11, 46.92, 22.23) mm, rotated rx -180 ry 0 rz -180 deg; joints [-18.787, 20.096, 41.054, 35.184, 33.982, -30.311]
  MoveL 479 to (240.11, 46.92, 22.23) mm, rotated rx -180 ry 0 rz -180 deg; joints [-18.787, 20.096, 41.054, 35.184, 33.982, -30.311]
  Call Extruder(426.47950)
  MoveL 480 to (240.15, 47.12, 22.23) mm, rotated rx 180 ry 0 rz -180 deg; joints [-18.807, 20.123, 41.016, 35.206, 34.001, -30.325]
  MoveL 481 to (240.15, 47.12, 22.23) mm, rotated rx 180 ry 0 rz -180 deg; joints [-18.807, 20.123, 41.016, 35.206, 34.001, -30.325]
  Call Extruder(426.71523)
  MoveL 482 to (240.2, 47.33, 22.22) mm, rotated rx 180 ry 0 rz 180 deg; joints [-18.827, 20.149, 40.979, 35.228, 34.02, -30.34]
  MoveL 483 to (240.2, 47.33, 22.22) mm, rotated rx 180 ry 0 rz 180 deg; joints [-18.827, 20.149, 40.979, 35.228, 34.02, -30.34]
  Call Extruder(426.97511)
  MoveL 484 to (240.24, 47.55, 22.22) mm, rotated rx -180 ry 0 rz 180 deg; joints [-18.85, 20.178, 40.938, 35.252, 34.04, -30.356]
  MoveL 485 to (240.24, 47.55, 22.22) mm, rotated rx -180 ry 0 rz 180 deg; joints [-18.85, 20.178, 40.938, 35.252, 34.04, -30.356]
  Call Extruder(427.25877)
  MoveL 486 to (240.29, 47.8, 22.22) mm, rotated rx 180 ry 0 rz 180 deg; joints [-18.874, 20.21, 40.893, 35.279, 34.063, -30.374]
  MoveL 487 to (240.29, 47.8, 22.22) mm, rotated rx 180 ry 0 rz 180 deg; joints [-18.874, 20.21, 40.893, 35.279, 34.063, -30.374]
  Call Extruder(427.54099)
  MoveL 488 to (240.34, 48.05, 22.23) mm, rotated rx 180 ry 0 rz 180 deg; joints [-18.899, 20.242, 40.849, 35.306, 34.086, -30.392]
  MoveL 489 to (240.34, 48.05, 22.23) mm, rotated rx 180 ry 0 rz 180 deg; joints [-18.899, 20.242, 40.849, 35.306, 34.086, -30.392]
  Call Extruder(427.82177)
  MoveL 490 to (240.39, 48.3, 22.23) mm, rotated rx 180 ry 0 rz 180 deg; joints [-18.923, 20.273, 40.804, 35.332, 34.109, -30.41]
  MoveL 491 to (240.39, 48.3, 22.23) mm, rotated rx 180 ry 0 rz 180 deg; joints [-18.923, 20.273, 40.804, 35.332, 34.109, -30.41]
  Call Extruder(428.10111)
  MoveL 492 to (240.44, 48.55, 22.23) mm, rotated rx 180 ry 0 rz 180 deg; joints [-18.948, 20.305, 40.76, 35.359, 34.132, -30.428]
  MoveL 493 to (240.44, 48.55, 22.23) mm, rotated rx 180 ry 0 rz 180 deg; joints [-18.948, 20.305, 40.76, 35.359, 34.132, -30.428]
  Call Extruder(428.37901)
  MoveL 494 to (240.49, 48.8, 22.23) mm, rotated rx 180 ry 0 rz 180 deg; joints [-18.973, 20.337, 40.715, 35.386, 34.155, -30.446]
  MoveL 495 to (240.49, 48.8, 22.23) mm, rotated rx 180 ry 0 rz 180 deg; joints [-18.973, 20.337, 40.715, 35.386, 34.155, -30.446]
  Call Extruder(428.65546)
  MoveL 496 to (240.54, 49.05, 22.22) mm, rotated rx 180 ry 0 rz 180 deg; joints [-18.997, 20.369, 40.67, 35.412, 34.178, -30.464]
  MoveL 497 to (240.54, 49.05, 22.22) mm, rotated rx 180 ry 0 rz 180 deg; joints [-18.997, 20.369, 40.67, 35.412, 34.178, -30.464]
  Call Extruder(428.96049)
  MoveL 498 to (240.59, 49.33, 22.22) mm, rotated rx 180 ry 0 rz 180 deg; joints [-19.025, 20.403, 40.622, 35.443, 34.203, -30.484]
  MoveL 499 to (240.59, 49.33, 22.22) mm, rotated rx 180 ry 0 rz 180 deg; joints [-19.025, 20.403, 40.622, 35.443, 34.203, -30.484]
  Call Extruder(429.29393)
  MoveL 500 to (240.64, 49.63, 22.23) mm, rotated rx 180 ry 0 rz 180 deg; joints [-19.055, 20.439, 40.571, 35.477, 34.231, -30.508]
  MoveL 501 to (240.64, 49.63, 22.23) mm, rotated rx 180 ry 0 rz 180 deg; joints [-19.055, 20.439, 40.571, 35.477, 34.231, -30.508]
  Call Extruder(429.62565)
  MoveL 502 to (240.69, 49.94, 22.22) mm, rotated rx -180 ry 0 rz 180 deg; joints [-19.086, 20.476, 40.52, 35.511, 34.259, -30.531]
  MoveL 503 to (240.69, 49.94, 22.22) mm, rotated rx -180 ry 0 rz 180 deg; joints [-19.086, 20.476, 40.52, 35.511, 34.259, -30.531]
  Call Extruder(429.95564)
  MoveL 504 to (240.73, 50.24, 22.22) mm, rotated rx -180 ry 0 rz 180 deg; joints [-19.116, 20.512, 40.468, 35.544, 34.286, -30.554]
  MoveL 505 to (240.73, 50.24, 22.22) mm, rotated rx -180 ry 0 rz 180 deg; joints [-19.116, 20.512, 40.468, 35.544, 34.286, -30.554]
  Call Extruder(430.28392)
  MoveL 506 to (240.78, 50.55, 22.23) mm, rotated rx 180 ry 0 rz 180 deg; joints [-19.146, 20.549, 40.416, 35.578, 34.314, -30.577]
  MoveL 507 to (240.78, 50.55, 22.23) mm, rotated rx 180 ry 0 rz 180 deg; joints [-19.146, 20.549, 40.416, 35.578, 34.314, -30.577]
  Call Extruder(430.61048)
  MoveL 508 to (240.83, 50.86, 22.23) mm, rotated rx 180 ry 0 rz 180 deg; joints [-19.177, 20.586, 40.364, 35.611, 34.342, -30.599]
  MoveL 509 to (240.83, 50.86, 22.23) mm, rotated rx 180 ry 0 rz 180 deg; joints [-19.177, 20.586, 40.364, 35.611, 34.342, -30.599]
  Call Extruder(430.97758)
  MoveL 510 to (240.88, 51.2, 22.23) mm, rotated rx -180 ry 0 rz 180 deg; joints [-19.212, 20.625, 40.308, 35.65, 34.373, -30.626]
  MoveL 511 to (240.88, 51.2, 22.23) mm, rotated rx -180 ry 0 rz 180 deg; joints [-19.212, 20.625, 40.308, 35.65, 34.373, -30.626]
  Call Extruder(431.38502)
  MoveL 512 to (240.92, 51.59, 22.23) mm, rotated rx 180 ry 0 rz 180 deg; joints [-19.251, 20.669, 40.247, 35.695, 34.408, -30.657]
  MoveL 513 to (240.92, 51.59, 22.23) mm, rotated rx 180 ry 0 rz 180 deg; joints [-19.251, 20.669, 40.247, 35.695, 34.408, -30.657]
  Call Extruder(431.79041)
  MoveL 514 to (240.97, 51.98, 22.22) mm, rotated rx -180 ry 0 rz 180 deg; joints [-19.29, 20.712, 40.186, 35.739, 34.442, -30.687]
  MoveL 515 to (240.97, 51.98, 22.22) mm, rotated rx -180 ry 0 rz 180 deg; joints [-19.29, 20.712, 40.186, 35.739, 34.442, -30.687]
  Call Extruder(432.19375)
  MoveL 516 to (241.02, 52.37, 22.22) mm, rotated rx 180 ry 0 rz 180 deg; joints [-19.329, 20.755, 40.124, 35.783, 34.477, -30.717]
  MoveL 517 to (241.02, 52.37, 22.22) mm, rotated rx 180 ry 0 rz 180 deg; joints [-19.329, 20.755, 40.124, 35.783, 34.477, -30.717]
  Call Extruder(432.59504)
  MoveL 518 to (241.06, 52.75, 22.22) mm, rotated rx 180 ry 0 rz 180 deg; joints [-19.368, 20.798, 40.063, 35.827, 34.511, -30.748]
  MoveL 519 to (241.06, 52.75, 22.22) mm, rotated rx 180 ry 0 rz 180 deg; joints [-19.368, 20.798, 40.063, 35.827, 34.511, -30.748]
  Call Extruder(433.20001)
  MoveL 520 to (241.11, 53.34, 22.22) mm, rotated rx -180 ry 0 rz 180 deg; joints [-19.428, 20.86, 39.976, 35.896, 34.563, -30.796]
  MoveL 521 to (241.11, 53.34, 22.22) mm, rotated rx -180 ry 0 rz 180 deg; joints [-19.428, 20.86, 39.976, 35.896, 34.563, -30.796]
  Call Extruder(433.80182)
  MoveL 522 to (241.15, 53.93, 22.23) mm, rotated rx 180 ry 0 rz 180 deg; joints [-19.488, 20.921, 39.89, 35.965, 34.614, -30.845]
  MoveL 523 to (241.15, 53.93, 22.23) mm, rotated rx 180 ry 0 rz 180 deg; joints [-19.488, 20.921, 39.89, 35.965, 34.614, -30.845]
  Call Extruder(434.40048)
  MoveL 524 to (241.2, 54.52, 22.22) mm, rotated rx -180 ry 0 rz -180 deg; joints [-19.548, 20.982, 39.802, 36.034, 34.666, -30.892]
  MoveL 525 to (241.2, 54.52, 22.22) mm, rotated rx -180 ry 0 rz -180 deg; joints [-19.548, 20.982, 39.802, 36.034, 34.666, -30.892]
  Call Extruder(435.57226)
  MoveL 526 to (241.25, 55.68, 22.22) mm, rotated rx 180 ry 0 rz 180 deg; joints [-19.668, 21.093, 39.644, 36.175, 34.766, -30.992]
  MoveL 527 to (241.25, 55.68, 22.22) mm, rotated rx 180 ry 0 rz 180 deg; joints [-19.668, 21.093, 39.644, 36.175, 34.766, -30.992]
  Call Extruder(437.02987)
  MoveL 528 to (241.29, 57.14, 22.23) mm, rotated rx -180 ry 0 rz -180 deg; joints [-19.819, 21.229, 39.45, 36.351, 34.89, -31.118]
  Call Extruder(522.92352)
  MoveL 529 to (241.29, 142.86, 22.22) mm, rotated rx -180 ry 0 rz -180 deg; joints [-28.232, 35.565, 16.466, 41.112, 46.007, -31.222]
  Call Extruder(523.79834)
  MoveL 530 to (241.27, 143.74, 22.22) mm, rotated rx 180 ry 0 rz 180 deg; joints [-28.313, 36.249, 15.225, 40.857, 46.47, -30.782]
  MoveL 531 to (241.27, 143.74, 22.22) mm, rotated rx 180 ry 0 rz 180 deg; joints [-28.313, 36.249, 15.225, 40.857, 46.47, -30.782]
  Call Extruder(524.97012)
  MoveL 532 to (241.22, 144.9, 22.22) mm, rotated rx 180 ry 0 rz -160 deg; joints [-22.789, 27.557, 29.957, 5.182, 32.592, -4.37]
  MoveL 533 to (241.23, 144.9, 22.22) mm, rotated rx 180 ry 0 rz -160 deg; joints [-22.789, 27.557, 29.957, 5.182, 32.592, -4.37]
  Call Extruder(525.85826)
  MoveL 534 to (241.18, 145.77, 22.22) mm, rotated rx 180 ry 0 rz -160 deg; joints [-22.877, 27.668, 29.782, 5.336, 32.663, -4.496]
  MoveL 535 to (241.18, 145.77, 22.22) mm, rotated rx 180 ry 0 rz -160 deg; joints [-22.877, 27.668, 29.782, 5.336, 32.663, -4.496]
  Call Extruder(526.46008)
  MoveL 536 to (241.13, 146.36, 22.22) mm, rotated rx 180 ry 0 rz -160 deg; joints [-22.937, 27.738, 29.672, 5.44, 32.708, -4.582]
  MoveL 537 to (241.13, 146.36, 22.22) mm, rotated rx 180 ry 0 rz -160 deg; joints [-22.937, 27.738, 29.672, 5.44, 32.708, -4.582]
  Call Extruder(527.06505)
  MoveL 538 to (241.09, 146.95, 22.23) mm, rotated rx 180 ry 0 rz -160 deg; joints [-22.996, 27.809, 29.56, 5.544, 32.754, -4.667]
  MoveL 539 to (241.09, 146.95, 22.23) mm, rotated rx 180 ry 0 rz -160 deg; joints [-22.996, 27.809, 29.56, 5.544, 32.754, -4.667]
  Call Extruder(527.56965)
  MoveL 540 to (241.04, 147.44, 22.22) mm, rotated rx 180 ry 0 rz -160 deg; joints [-23.046, 27.865, 29.471, 5.631, 32.79, -4.738]
  MoveL 541 to (241.04, 147.44, 22.22) mm, rotated rx 180 ry 0 rz -160 deg; joints [-23.046, 27.865, 29.471, 5.631, 32.79, -4.738]
  Call Extruder(527.97299)
  MoveL 542 to (240.99, 147.83, 22.22) mm, rotated rx 180 ry 0 rz -160 deg; joints [-23.086, 27.906, 29.405, 5.701, 32.818, -4.795]
  MoveL 543 to (240.99, 147.83, 22.22) mm, rotated rx 180 ry 0 rz -160 deg; joints [-23.086, 27.906, 29.405, 5.701, 32.818, -4.795]
  Call Extruder(528.37839)
  MoveL 544 to (240.95, 148.22, 22.22) mm, rotated rx 180 ry 0 rz -160 deg; joints [-23.126, 27.948, 29.339, 5.77, 32.845, -4.852]
  MoveL 545 to (240.95, 148.22, 22.22) mm, rotated rx 180 ry 0 rz -160 deg; joints [-23.126, 27.948, 29.339, 5.77, 32.845, -4.852]
  Call Extruder(528.78583)
  MoveL 546 to (240.9, 148.6, 22.22) mm, rotated rx -180 ry 0 rz -160 deg; joints [-23.166, 27.99, 29.272, 5.839, 32.873, -4.909]
  MoveL 547 to (240.9, 148.6, 22.22) mm, rotated rx -180 ry 0 rz -160 deg; joints [-23.166, 27.99, 29.272, 5.839, 32.873, -4.909]
  Call Extruder(529.19532)
  MoveL 548 to (240.86, 148.99, 22.23) mm, rotated rx -180 ry 0 rz -160 deg; joints [-23.206, 28.033, 29.205, 5.909, 32.902, -4.966]
  MoveL 549 to (240.86, 148.99, 22.23) mm, rotated rx -180 ry 0 rz -160 deg; joints [-23.206, 28.033, 29.205, 5.909, 32.902, -4.966]
  Call Extruder(529.52188)
  MoveL 550 to (240.81, 149.3, 22.23) mm, rotated rx 180 ry 0 rz -160 deg; joints [-23.237, 28.062, 29.158, 5.964, 32.922, -5.012]
  MoveL 551 to (240.81, 149.3, 22.23) mm, rotated rx 180 ry 0 rz -160 deg; joints [-23.237, 28.062, 29.158, 5.964, 32.922, -5.012]
  Call Extruder(529.85015)
  MoveL 552 to (240.76, 149.6, 22.22) mm, rotated rx 180 ry 0 rz -160 deg; joints [-23.269, 28.092, 29.111, 6.02, 32.942, -5.058]
  MoveL 553 to (240.76, 149.6, 22.22) mm, rotated rx 180 ry 0 rz -160 deg; joints [-23.269, 28.092, 29.111, 6.02, 32.942, -5.058]
  Call Extruder(530.18015)
  MoveL 554 to (240.71, 149.91, 22.23) mm, rotated rx -180 ry 0 rz -160 deg; joints [-23.301, 28.121, 29.064, 6.076, 32.962, -5.103]
  MoveL 555 to (240.71, 149.91, 22.23) mm, rotated rx -180 ry 0 rz -160 deg; joints [-23.301, 28.121, 29.064, 6.076, 32.962, -5.103]
  Call Extruder(530.51186)
  MoveL 556 to (240.66, 150.21, 22.23) mm, rotated rx 180 ry 0 rz -160 deg; joints [-23.333, 28.151, 29.017, 6.131, 32.982, -5.149]
  MoveL 557 to (240.66, 150.21, 22.23) mm, rotated rx 180 ry 0 rz -160 deg; joints [-23.333, 28.151, 29.017, 6.131, 32.982, -5.149]
  Call Extruder(530.84529)
  MoveL 558 to (240.61, 150.52, 22.23) mm, rotated rx 180 ry 0 rz -160 deg; joints [-23.365, 28.181, 28.969, 6.187, 33.003, -5.194]
  MoveL 559 to (240.61, 150.52, 22.23) mm, rotated rx 180 ry 0 rz -160 deg; joints [-23.365, 28.181, 28.969, 6.187, 33.003, -5.194]
  Call Extruder(531.18045)
  MoveL 560 to (240.57, 150.83, 22.22) mm, rotated rx 180 ry 0 rz -160 deg; joints [-23.397, 28.211, 28.922, 6.242, 33.023, -5.24]
  MoveL 561 to (240.57, 150.83, 22.22) mm, rotated rx 180 ry 0 rz -160 deg; joints [-23.397, 28.211, 28.922, 6.242, 33.023, -5.24]
  Call Extruder(531.45690)
  MoveL 562 to (240.52, 151.08, 22.23) mm, rotated rx 180 ry 0 rz -160 deg; joints [-23.423, 28.232, 28.888, 6.288, 33.038, -5.278]
  MoveL 563 to (240.52, 151.08, 22.23) mm, rotated rx 180 ry 0 rz -160 deg; joints [-23.423, 28.232, 28.888, 6.288, 33.038, -5.278]
  Call Extruder(531.73480)
  MoveL 564 to (240.47, 151.32, 22.22) mm, rotated rx 180 ry 0 rz -160 deg; joints [-23.45, 28.252, 28.855, 6.334, 33.053, -5.316]
  MoveL 565 to (240.47, 151.32, 22.22) mm, rotated rx 180 ry 0 rz -160 deg; joints [-23.45, 28.252, 28.855, 6.334, 33.053, -5.316]
  Call Extruder(532.01414)
  MoveL 566 to (240.42, 151.57, 22.22) mm, rotated rx 180 ry 0 rz -160 deg; joints [-23.476, 28.273, 28.822, 6.38, 33.067, -5.353]
  MoveL 567 to (240.42, 151.57, 22.22) mm, rotated rx 180 ry 0 rz -160 deg; joints [-23.476, 28.273, 28.822, 6.38, 33.067, -5.353]
  Call Extruder(532.29492)
  MoveL 568 to (240.37, 151.82, 22.22) mm, rotated rx 180 ry 0 rz -160 deg; joints [-23.503, 28.295, 28.788, 6.426, 33.082, -5.391]
  MoveL 569 to (240.37, 151.82, 22.22) mm, rotated rx 180 ry 0 rz -160 deg; joints [-23.503, 28.295, 28.788, 6.426, 33.082, -5.391]
  Call Extruder(532.57714)
  MoveL 570 to (240.32, 152.07, 22.22) mm, rotated rx 180 ry 0 rz -160 deg; joints [-23.529, 28.316, 28.754, 6.472, 33.097, -5.429]
  MoveL 571 to (240.32, 152.07, 22.22) mm, rotated rx 180 ry 0 rz -160 deg; joints [-23.529, 28.316, 28.754, 6.472, 33.097, -5.429]
  Call Extruder(532.86081)
  MoveL 572 to (240.27, 152.32, 22.22) mm, rotated rx 180 ry 0 rz -160 deg; joints [-23.555, 28.337, 28.72, 6.518, 33.113, -5.466]
  MoveL 573 to (240.27, 152.32, 22.22) mm, rotated rx 180 ry 0 rz -160 deg; joints [-23.555, 28.337, 28.72, 6.518, 33.113, -5.466]
  Call Extruder(533.14591)
  MoveL 574 to (240.22, 152.57, 22.22) mm, rotated rx 180 ry 0 rz -160 deg; joints [-23.582, 28.359, 28.686, 6.564, 33.128, -5.504]
  MoveL 575 to (240.22, 152.57, 22.22) mm, rotated rx 180 ry 0 rz -160 deg; joints [-23.582, 28.359, 28.686, 6.564, 33.128, -5.504]
  Call Extruder(533.38165)
  MoveL 576 to (240.17, 152.77, 22.22) mm, rotated rx 180 ry 0 rz -160 deg; joints [-23.603, 28.375, 28.66, 6.602, 33.139, -5.535]
  MoveL 577 to (240.17, 152.77, 22.22) mm, rotated rx 180 ry 0 rz -160 deg; joints [-23.603, 28.375, 28.66, 6.602, 33.139, -5.535]
  Call Extruder(533.61845)
  MoveL 578 to (240.13, 152.98, 22.23) mm, rotated rx -180 ry 0 rz -160 deg; joints [-23.625, 28.391, 28.634, 6.64, 33.151, -5.566]
  MoveL 579 to (240.13, 152.98, 22.23) mm, rotated rx -180 ry 0 rz -160 deg; joints [-23.625, 28.391, 28.634, 6.64, 33.151, -5.566]
  Call Extruder(533.85633)
  MoveL 580 to (240.08, 153.18, 22.22) mm, rotated rx 180 ry 0 rz -160 deg; joints [-23.647, 28.407, 28.608, 6.678, 33.163, -5.598]
  MoveL 581 to (240.08, 153.18, 22.22) mm, rotated rx 180 ry 0 rz -160 deg; joints [-23.647, 28.407, 28.608, 6.678, 33.163, -5.598]
  Call Extruder(534.09527)
  MoveL 582 to (240.04, 153.39, 22.22) mm, rotated rx 180 ry 0 rz -160 deg; joints [-23.669, 28.424, 28.582, 6.715, 33.175, -5.629]
  MoveL 583 to (240.04, 153.39, 22.22) mm, rotated rx 180 ry 0 rz -160 deg; joints [-23.669, 28.424, 28.582, 6.715, 33.175, -5.629]
  Call Extruder(534.34924)
  MoveL 584 to (239.98, 153.6, 22.23) mm, rotated rx 180 ry 0 rz -160 deg; joints [-23.692, 28.438, 28.56, 6.756, 33.185, -5.662]
  MoveL 585 to (239.98, 153.6, 22.23) mm, rotated rx 180 ry 0 rz -160 deg; joints [-23.692, 28.438, 28.56, 6.756, 33.185, -5.662]
  Call Extruder(534.61883)
  MoveL 586 to (239.92, 153.82, 22.22) mm, rotated rx 180 ry 0 rz -160 deg; joints [-23.717, 28.449, 28.542, 6.8, 33.194, -5.698]
  MoveL 587 to (239.92, 153.82, 22.22) mm, rotated rx 180 ry 0 rz -160 deg; joints [-23.717, 28.449, 28.542, 6.8, 33.194, -5.698]
  Call Extruder(534.88976)
  MoveL 588 to (239.85, 154.05, 22.22) mm, rotated rx 180 ry 0 rz -160 deg; joints [-23.741, 28.46, 28.525, 6.843, 33.203, -5.734]
  MoveL 589 to (239.85, 154.05, 22.22) mm, rotated rx 180 ry 0 rz -160 deg; joints [-23.741, 28.46, 28.525, 6.843, 33.203, -5.734]
  Call Extruder(535.16202)
  MoveL 590 to (239.78, 154.27, 22.22) mm, rotated rx -180 ry 0 rz -160 deg; joints [-23.766, 28.471, 28.506, 6.887, 33.212, -5.77]
  MoveL 591 to (239.78, 154.27, 22.22) mm, rotated rx -180 ry 0 rz -160 deg; joints [-23.766, 28.471, 28.506, 6.887, 33.212, -5.77]
  Call Extruder(535.43561)
  MoveL 592 to (239.71, 154.5, 22.22) mm, rotated rx 180 ry 0 rz -160 deg; joints [-23.791, 28.482, 28.488, 6.93, 33.222, -5.806]
  MoveL 593 to (239.71, 154.5, 22.22) mm, rotated rx 180 ry 0 rz -160 deg; joints [-23.791, 28.482, 28.488, 6.93, 33.222, -5.806]
  Call Extruder(535.66881)
  MoveL 594 to (239.65, 154.68, 22.22) mm, rotated rx 180 ry 0 rz -160 deg; joints [-23.811, 28.49, 28.476, 6.967, 33.229, -5.837]
  MoveL 595 to (239.65, 154.68, 22.22) mm, rotated rx 180 ry 0 rz -160 deg; joints [-23.811, 28.49, 28.476, 6.967, 33.229, -5.837]
  Call Extruder(535.90306)
  MoveL 596 to (239.59, 154.87, 22.22) mm, rotated rx -180 ry 0 rz -160 deg; joints [-23.832, 28.499, 28.462, 7.005, 33.236, -5.868]
  MoveL 597 to (239.59, 154.87, 22.22) mm, rotated rx -180 ry 0 rz -160 deg; joints [-23.832, 28.499, 28.462, 7.005, 33.236, -5.868]
  Call Extruder(536.13835)
  MoveL 598 to (239.53, 155.06, 22.23) mm, rotated rx -180 ry 0 rz -160 deg; joints [-23.853, 28.506, 28.45, 7.042, 33.242, -5.898]
  MoveL 599 to (239.53, 155.06, 22.23) mm, rotated rx -180 ry 0 rz -160 deg; joints [-23.853, 28.506, 28.45, 7.042, 33.242, -5.898]
  Call Extruder(536.37470)
  MoveL 600 to (239.47, 155.25, 22.22) mm, rotated rx 180 ry 0 rz -160 deg; joints [-23.874, 28.515, 28.437, 7.079, 33.249, -5.929]
  MoveL 601 to (239.47, 155.25, 22.22) mm, rotated rx 180 ry 0 rz -160 deg; joints [-23.874, 28.515, 28.437, 7.079, 33.249, -5.929]
  Call Extruder(536.61210)
  MoveL 602 to (239.41, 155.44, 22.22) mm, rotated rx -180 ry 0 rz -160 deg; joints [-23.895, 28.523, 28.424, 7.116, 33.256, -5.96]
  MoveL 603 to (239.41, 155.44, 22.22) mm, rotated rx -180 ry 0 rz -160 deg; joints [-23.895, 28.523, 28.424, 7.116, 33.256, -5.96]
  Call Extruder(536.99230)
  MoveL 604 to (239.29, 155.73, 22.22) mm, rotated rx 180 ry 0 rz -160 deg; joints [-23.929, 28.526, 28.419, 7.176, 33.262, -6.01]
  MoveL 605 to (239.29, 155.73, 22.22) mm, rotated rx 180 ry 0 rz -160 deg; joints [-23.929, 28.526, 28.419, 7.176, 33.262, -6.01]
  Call Extruder(537.37429)
  MoveL 606 to (239.16, 156.02, 22.22) mm, rotated rx 180 ry 0 rz -160 deg; joints [-23.962, 28.529, 28.414, 7.237, 33.267, -6.06]
  MoveL 607 to (239.16, 156.02, 22.22) mm, rotated rx 180 ry 0 rz -160 deg; joints [-23.962, 28.529, 28.414, 7.237, 33.267, -6.06]
  Call Extruder(537.73076)
  MoveL 608 to (239.05, 156.29, 22.23) mm, rotated rx 180 ry 0 rz -160 deg; joints [-23.993, 28.531, 28.41, 7.293, 33.272, -6.107]
  MoveL 609 to (239.05, 156.29, 22.23) mm, rotated rx 180 ry 0 rz -160 deg; joints [-23.993, 28.531, 28.41, 7.293, 33.272, -6.107]
  Call Extruder(538.06143)
  MoveL 610 to (238.94, 156.54, 22.22) mm, rotated rx 180 ry 0 rz -160 deg; joints [-24.022, 28.533, 28.408, 7.345, 33.276, -6.151]
  MoveL 611 to (238.94, 156.54, 22.22) mm, rotated rx 180 ry 0 rz -160 deg; joints [-24.022, 28.533, 28.408, 7.345, 33.276, -6.151]
  Call Extruder(538.39353)
  MoveL 612 to (238.84, 156.79, 22.22) mm, rotated rx 180 ry 0 rz -160 deg; joints [-24.051, 28.534, 28.405, 7.397, 33.28, -6.194]
  MoveL 613 to (238.84, 156.79, 22.22) mm, rotated rx 180 ry 0 rz -160 deg; joints [-24.051, 28.534, 28.405, 7.397, 33.28, -6.194]
  Call Extruder(538.82540)
  MoveL 614 to (238.66, 157.09, 22.22) mm, rotated rx 180 ry 0 rz -160 deg; joints [-24.088, 28.52, 28.428, 7.466, 33.275, -6.252]
  MoveL 615 to (238.66, 157.09, 22.22) mm, rotated rx 180 ry 0 rz -160 deg; joints [-24.088, 28.52, 28.428, 7.466, 33.275, -6.252]
  Call Extruder(539.25912)
  MoveL 616 to (238.49, 157.4, 22.23) mm, rotated rx -180 ry 0 rz -160 deg; joints [-24.125, 28.505, 28.452, 7.535, 33.271, -6.311]
  MoveL 617 to (238.49, 157.4, 22.23) mm, rotated rx -180 ry 0 rz -160 deg; joints [-24.125, 28.505, 28.452, 7.535, 33.271, -6.311]
  Call Extruder(539.69468)
  MoveL 618 to (238.31, 157.7, 22.23) mm, rotated rx 180 ry 0 rz -160 deg; joints [-24.162, 28.491, 28.474, 7.604, 33.266, -6.369]
  MoveL 619 to (238.31, 157.7, 22.23) mm, rotated rx 180 ry 0 rz -160 deg; joints [-24.162, 28.491, 28.474, 7.604, 33.266, -6.369]
  Call Extruder(540.13207)
  MoveL 620 to (238.14, 158.01, 22.22) mm, rotated rx 180 ry 0 rz -160 deg; joints [-24.199, 28.477, 28.497, 7.672, 33.262, -6.427]
  MoveL 621 to (238.14, 158.01, 22.22) mm, rotated rx 180 ry 0 rz -160 deg; joints [-24.199, 28.477, 28.497, 7.672, 33.262, -6.427]
  Call Extruder(540.50882)
  MoveL 622 to (237.96, 158.25, 22.22) mm, rotated rx -180 ry 0 rz -160 deg; joints [-24.231, 28.453, 28.536, 7.732, 33.251, -6.478]
  MoveL 623 to (237.96, 158.25, 22.22) mm, rotated rx -180 ry 0 rz -160 deg; joints [-24.231, 28.453, 28.536, 7.732, 33.251, -6.478]
  Call Extruder(541.20873)
  MoveL 624 to (237.63, 158.7, 22.22) mm, rotated rx 180 ry 0 rz -160 deg; joints [-24.289, 28.408, 28.608, 7.843, 33.231, -6.573]
  MoveL 625 to (237.63, 158.7, 22.22) mm, rotated rx 180 ry 0 rz -160 deg; joints [-24.289, 28.408, 28.608, 7.843, 33.231, -6.573]
  Call Extruder(541.91145)
  MoveL 626 to (237.3, 159.15, 22.22) mm, rotated rx 180 ry 0 rz -160 deg; joints [-24.347, 28.363, 28.679, 7.954, 33.211, -6.668]
  Call Extruder(543.65031)
  MoveL 627 to (236.39, 160.19, 22.22) mm, rotated rx 180 ry 0 rz -160 deg; joints [-24.487, 28.205, 28.931, 8.229, 33.135, -6.905]
  Call Extruder(545.38913)
  MoveL 628 to (235.35, 161.1, 22.23) mm, rotated rx 180 ry 0 rz -160 deg; joints [-24.621, 27.987, 29.278, 8.502, 33.024, -7.144]
  Call Extruder(545.74051)
  MoveL 629 to (235.13, 161.27, 22.23) mm, rotated rx 180 ry 0 rz -160 deg; joints [-24.647, 27.934, 29.361, 8.556, 32.997, -7.192]
  MoveL 630 to (235.13, 161.27, 22.23) mm, rotated rx 180 ry 0 rz -160 deg; joints [-24.647, 27.934, 29.361, 8.556, 32.997, -7.192]
  Call Extruder(546.44047)
  MoveL 631 to (234.68, 161.59, 22.23) mm, rotated rx 180 ry 0 rz -160 deg; joints [-24.699, 27.83, 29.525, 8.664, 32.944, -7.287]
  MoveL 632 to (234.68, 161.59, 22.23) mm, rotated rx 180 ry 0 rz -160 deg; joints [-24.699, 27.83, 29.525, 8.664, 32.944, -7.287]
  Call Extruder(547.13763)
  MoveL 633 to (234.23, 161.92, 22.22) mm, rotated rx 180 ry 0 rz -160 deg; joints [-24.751, 27.728, 29.688, 8.773, 32.891, -7.384]
  MoveL 634 to (234.23, 161.92, 22.22) mm, rotated rx 180 ry 0 rz -160 deg; joints [-24.751, 27.728, 29.688, 8.773, 32.891, -7.384]
  Call Extruder(547.38444)
  MoveL 635 to (234.05, 162.02, 22.22) mm, rotated rx 180 ry 0 rz -160 deg; joints [-24.768, 27.685, 29.755, 8.81, 32.869, -7.417]
  MoveL 636 to (234.05, 162.02, 22.22) mm, rotated rx 180 ry 0 rz -160 deg; joints [-24.768, 27.685, 29.755, 8.81, 32.869, -7.417]
  Call Extruder(547.82000)
  MoveL 637 to (233.75, 162.2, 22.23) mm, rotated rx 180 ry 0 rz -160 deg; joints [-24.799, 27.609, 29.875, 8.877, 32.83, -7.476]
  MoveL 638 to (233.75, 162.2, 22.23) mm, rotated rx 180 ry 0 rz -160 deg; joints [-24.799, 27.609, 29.875, 8.877, 32.83, -7.476]
  Call Extruder(548.25372)
  MoveL 639 to (233.45, 162.37, 22.23) mm, rotated rx 180 ry 0 rz -160 deg; joints [-24.829, 27.534, 29.993, 8.943, 32.791, -7.536]
  MoveL 640 to (233.45, 162.37, 22.23) mm, rotated rx 180 ry 0 rz -160 deg; joints [-24.829, 27.534, 29.993, 8.943, 32.791, -7.536]
  Call Extruder(548.68559)
  MoveL 641 to (233.14, 162.55, 22.22) mm, rotated rx 180 ry 0 rz -160 deg; joints [-24.86, 27.46, 30.11, 9.009, 32.753, -7.595]
  MoveL 642 to (233.14, 162.55, 22.22) mm, rotated rx 180 ry 0 rz -160 deg; joints [-24.86, 27.46, 30.11, 9.009, 32.753, -7.595]
  Call Extruder(549.06597)
  MoveL 643 to (232.87, 162.69, 22.22) mm, rotated rx 180 ry 0 rz -160 deg; joints [-24.886, 27.389, 30.221, 9.067, 32.716, -7.647]
  MoveL 644 to (232.87, 162.69, 22.22) mm, rotated rx 180 ry 0 rz -160 deg; joints [-24.886, 27.389, 30.221, 9.067, 32.716, -7.647]
  Call Extruder(549.39656)
  MoveL 645 to (232.62, 162.8, 22.22) mm, rotated rx 180 ry 0 rz -160 deg; joints [-24.908, 27.324, 30.324, 9.116, 32.682, -7.692]
  MoveL 646 to (232.62, 162.8, 22.22) mm, rotated rx 180 ry 0 rz -160 deg; joints [-24.908, 27.324, 30.324, 9.116, 32.682, -7.692]
  Call Extruder(549.72573)
  MoveL 647 to (232.37, 162.9, 22.23) mm, rotated rx 180 ry 0 rz -160 deg; joints [-24.929, 27.258, 30.427, 9.165, 32.648, -7.736]
  MoveL 648 to (232.37, 162.9, 22.23) mm, rotated rx 180 ry 0 rz -160 deg; joints [-24.929, 27.258, 30.427, 9.165, 32.648, -7.736]
  Call Extruder(550.10778)
  MoveL 649 to (232.08, 163.03, 22.22) mm, rotated rx 180 ry 0 rz -160 deg; joints [-24.954, 27.181, 30.549, 9.221, 32.608, -7.787]
  MoveL 650 to (232.08, 163.03, 22.22) mm, rotated rx 180 ry 0 rz -160 deg; joints [-24.954, 27.181, 30.549, 9.221, 32.608, -7.787]
  Call Extruder(550.48803)
  MoveL 651 to (231.78, 163.15, 22.22) mm, rotated rx 180 ry 0 rz -160 deg; joints [-24.979, 27.104, 30.669, 9.278, 32.569, -7.839]
  MoveL 652 to (231.78, 163.15, 22.22) mm, rotated rx 180 ry 0 rz -160 deg; joints [-24.979, 27.104, 30.669, 9.278, 32.569, -7.839]
  Call Extruder(550.79572)
  MoveL 653 to (231.54, 163.24, 22.22) mm, rotated rx 180 ry 0 rz -160 deg; joints [-24.999, 27.04, 30.769, 9.323, 32.536, -7.88]
  MoveL 654 to (231.54, 163.24, 22.22) mm, rotated rx 180 ry 0 rz -160 deg; joints [-24.999, 27.04, 30.769, 9.323, 32.536, -7.88]
  Call Extruder(551.03204)
  MoveL 655 to (231.35, 163.3, 22.22) mm, rotated rx 180 ry 0 rz -160 deg; joints [-25.013, 26.988, 30.849, 9.358, 32.509, -7.912]
  MoveL 656 to (231.35, 163.3, 22.22) mm, rotated rx 180 ry 0 rz -160 deg; joints [-25.013, 26.988, 30.849, 9.358, 32.509, -7.912]
  Call Extruder(551.26731)
  MoveL 657 to (231.17, 163.36, 22.22) mm, rotated rx -180 ry 0 rz -160 deg; joints [-25.028, 26.937, 30.929, 9.392, 32.483, -7.943]
  MoveL 658 to (231.17, 163.36, 22.22) mm, rotated rx -180 ry 0 rz -160 deg; joints [-25.028, 26.937, 30.929, 9.392, 32.483, -7.943]
  Call Extruder(551.50153)
  MoveL 659 to (230.98, 163.42, 22.23) mm, rotated rx 180 ry 0 rz -160 deg; joints [-25.042, 26.886, 31.009, 9.426, 32.457, -7.974]
  MoveL 660 to (230.98, 163.42, 22.23) mm, rotated rx 180 ry 0 rz -160 deg; joints [-25.042, 26.886, 31.009, 9.426, 32.457, -7.974]
  Call Extruder(551.73470)
  MoveL 661 to (230.79, 163.48, 22.23) mm, rotated rx 180 ry 0 rz -160 deg; joints [-25.056, 26.835, 31.089, 9.46, 32.431, -8.005]
  MoveL 662 to (230.79, 163.48, 22.23) mm, rotated rx 180 ry 0 rz -160 deg; joints [-25.056, 26.835, 31.089, 9.46, 32.431, -8.005]
  Call Extruder(551.98757)
  MoveL 663 to (230.58, 163.55, 22.23) mm, rotated rx 180 ry 0 rz -160 deg; joints [-25.072, 26.779, 31.175, 9.497, 32.402, -8.039]
  MoveL 664 to (230.58, 163.55, 22.23) mm, rotated rx 180 ry 0 rz -160 deg; joints [-25.072, 26.779, 31.175, 9.497, 32.402, -8.039]
  Call Extruder(552.25988)
  MoveL 665 to (230.36, 163.61, 22.23) mm, rotated rx -180 ry 0 rz -160 deg; joints [-25.089, 26.718, 31.27, 9.536, 32.371, -8.076]
  MoveL 666 to (230.36, 163.61, 22.23) mm, rotated rx -180 ry 0 rz -160 deg; joints [-25.089, 26.718, 31.27, 9.536, 32.371, -8.076]
  Call Extruder(552.53085)
  MoveL 667 to (230.14, 163.68, 22.22) mm, rotated rx 180 ry 0 rz -160 deg; joints [-25.106, 26.658, 31.364, 9.576, 32.341, -8.112]
